LIN {X 0,Y 573.249,Z 308.076,A -85,B 0,C 180,E1 -2303.077,E2 -2303.077} C_VEL
LIN {X 0,Y 573.266,Z 308.08,A -85,B 0,C 180,E1 -2305.671,E2 -2305.671} C_VEL
LIN {X 0,Y 573.24,Z 308.077,A -85,B 0,C 180,E1 -2308.184,E2 -2308.184} C_VEL
LIN {X 0,Y 573.229,Z 308.083,A -85,B 0,C 180,E1 -2310.632,E2 -2310.632} C_VEL
LIN {X 0,Y 573.245,Z 308.077,A -85,B 0,C 180,E1 -2313.809,E2 -2313.809} C_VEL
LIN {X 0,Y 573.224,Z 308.085,A -85,B 0,C 180,E1 -2316.134,E2 -2316.134} C_VEL
LIN {X 0,Y 573.253,Z 308.079,A -85,B 0,C 180,E1 -2319.174,E2 -2319.174} C_VEL
LIN {X 0,Y 573.227,Z 308.083,A -85,B 0,C 180,E1 -2321.411,E2 -2321.411} C_VEL
LIN {X 0,Y 573.228,Z 308.079,A -85,B 0,C 180,E1 -2323.621,E2 -2323.621} C_VEL
LIN {X 0,Y 573.243,Z 308.078,A -85,B 0,C 180,E1 -2325.806,E2 -2325.806} C_VEL
LIN {X 0,Y 573.251,Z 308.075,A -85,B 0,C 180,E1 -2328.745,E2 -2328.745} C_VEL
LIN {X 0,Y 573.299,Z 308.076,A -85,B 0,C 180,E1 -2331.541,E2 -2331.541} C_VEL
LIN {X 0,Y 573.299,Z 308.071,A -85,B 0,C 180,E1 -2334.372,E2 -2334.372} C_VEL
LIN {X 0,Y 573.306,Z 308.071,A -85,B 0,C 180,E1 -2337.892,E2 -2337.892} C_VEL
LIN {X 0,Y 573.301,Z 308.069,A -85,B 0,C 180,E1 -2340.702,E2 -2340.702} C_VEL
LIN {X 0,Y 573.286,Z 308.071,A -85,B 0,C 180,E1 -2342.811,E2 -2342.811} C_VEL
LIN {X 0,Y 573.299,Z 308.071,A -85,B 0,C 180,E1 -2345.628,E2 -2345.628} C_VEL
LIN {X 0,Y 573.299,Z 308.076,A -85,B 0,C 180,E1 -2348.459,E2 -2348.459} C_VEL
LIN {X 0,Y 573.26,Z 308.075,A -85,B 0,C 180,E1 -2351.312,E2 -2351.312} C_VEL
LIN {X 0,Y 573.254,Z 308.075,A -85,B 0,C 180,E1 -2354.419,E2 -2354.419} C_VEL
LIN {X 0,Y 573.248,Z 308.083,A -85,B 0,C 180,E1 -2357.112,E2 -2357.112} C_VEL
LIN {X 0,Y 573.249,Z 308.077,A -85,B 0,C 180,E1 -2360.077,E2 -2360.077} C_VEL
LIN {X 0,Y 573.23,Z 308.085,A -85,B 0,C 180,E1 -2362.338,E2 -2362.338} C_VEL
LIN {X 0,Y 573.242,Z 308.078,A -85,B 0,C 180,E1 -2364.396,E2 -2364.396} C_VEL
LIN {X 0,Y 572.612,Z 308.156,A -85,B 0,C 180,E1 -2364.982,E2 -2364.982} C_VEL
LIN {X 0,Y 569.758,Z 308.518,A -85,B 0,C 180,E1 -2365.933,E2 -2365.933} C_VEL
LIN {X 0,Y 567.31,Z 308.826,A -85,B 0,C 180,E1 -2366.699,E2 -2366.699} C_VEL
LIN {X 0,Y 566.241,Z 308.956,A -85,B 0,C 180,E1 -2367.29,E2 -2367.29} C_VEL
LIN {X 0,Y 566.146,Z 308.965,A -85,B 0,C 180,E1 -2367.49,E2 -2367.49} C_VEL
LIN {X 0,Y 566.162,Z 308.959,A -85,B 0,C 180,E1 -2369.771,E2 -2369.771} C_VEL
LIN {X 0,Y 566.2,Z 308.959,A -85,B 0,C 180,E1 -2372.432,E2 -2372.432} C_VEL
LIN {X 0,Y 566.205,Z 308.954,A -85,B 0,C 180,E1 -2374.995,E2 -2374.995} C_VEL
LIN {X 0,Y 566.189,Z 308.96,A -85,B 0,C 180,E1 -2377.462,E2 -2377.462} C_VEL
LIN {X 0,Y 566.2,Z 308.954,A -85,B 0,C 180,E1 -2380.2,E2 -2380.2} C_VEL
LIN {X 0,Y 566.175,Z 308.961,A -85,B 0,C 180,E1 -2383.057,E2 -2383.057} C_VEL
LIN {X 0,Y 566.194,Z 308.958,A -85,B 0,C 180,E1 -2386.05,E2 -2386.05} C_VEL
LIN {X 0,Y 566.208,Z 308.953,A -85,B 0,C 180,E1 -2388.865,E2 -2388.865} C_VEL
LIN {X 0,Y 566.184,Z 308.961,A -85,B 0,C 180,E1 -2391.638,E2 -2391.638} C_VEL
LIN {X 0,Y 566.132,Z 308.964,A -85,B 0,C 180,E1 -2394.307,E2 -2394.307} C_VEL
LIN {X 0,Y 566.172,Z 309.762,A -85,B 0,C 180,E1 -2395.181,E2 -2395.181} C_VEL
LIN {X 0,Y 566.158,Z 313.905,A -85,B 0,C 180,E1 -2397.74,E2 -2397.74} C_VEL
LIN {X 0,Y 566.063,Z 318.167,A -85,B 0,C 180,E1 -2400.354,E2 -2400.354} C_VEL
LIN {X 0,Y 566.044,Z 322,A -85,B 0,C 180,E1 -2402.653,E2 -2402.653} C_VEL
LIN {X 0,Y 566.04,Z 326.033,A -85,B 0,C 180,E1 -2405.031,E2 -2405.031} C_VEL
LIN {X 0,Y 565.976,Z 330.049,A -85,B 0,C 180,E1 -2407.361,E2 -2407.361} C_VEL
LIN {X 0,Y 565.93,Z 334.103,A -85,B 0,C 180,E1 -2409.653,E2 -2409.653} C_VEL
LIN {X 0,Y 565.903,Z 338.25,A -85,B 0,C 180,E1 -2411.913,E2 -2411.913} C_VEL
LIN {X 0,Y 565.913,Z 343.78,A -85,B 0,C 180,E1 -2414.883,E2 -2414.883} C_VEL
LIN {X 0,Y 565.889,Z 348.532,A -85,B 0,C 180,E1 -2417.402,E2 -2417.402} C_VEL
LIN {X 0,Y 566.917,Z 355.474,A -85,B 0,C 180,E1 -2417.585,E2 -2417.585} C_VEL
LIN {X 0,Y 566.768,Z 368.5,A -85,B 0,C 180,E1 -2417.968,E2 -2417.968} C_VEL
LIN {X 0,Y 566.608,Z 381.072,A -85,B 0,C 180,E1 -2418.491,E2 -2418.491} C_VEL
LIN {X 0,Y 566.531,Z 392.345,A -85,B 0,C 180,E1 -2419.114,E2 -2419.114} C_VEL
LIN {X 0,Y 566.404,Z 403.688,A -85,B 0,C 180,E1 -2419.906,E2 -2419.906} C_VEL
LIN {X 0,Y 566.255,Z 413.063,A -85,B 0,C 180,E1 -2420.715,E2 -2420.715} C_VEL
LIN {X 0,Y 566.158,Z 421.62,A -85,B 0,C 180,E1 -2421.613,E2 -2421.613} C_VEL
LIN {X 0,Y 566.063,Z 429.931,A -85,B 0,C 180,E1 -2422.689,E2 -2422.689} C_VEL
LIN {X 0,Y 565.988,Z 436.626,A -85,B 0,C 180,E1 -2423.763,E2 -2423.763} C_VEL
LIN {X 0,Y 565.877,Z 442.766,A -85,B 0,C 180,E1 -2425.013,E2 -2425.013} C_VEL
LIN {X 0,Y 565.926,Z 446.755,A -85,B 0,C 180,E1 -2426.084,E2 -2426.084} C_VEL
LIN {X 0,Y 565.877,Z 449.703,A -85,B 0,C 180,E1 -2427.153,E2 -2427.153} C_VEL
LIN {X 0,Y 565.841,Z 451.128,A -85,B 0,C 180,E1 -2427.865,E2 -2427.865} C_VEL
LIN {X 0,Y 565.841,Z 452.756,A -85,B 0,C 180,E1 -2429.289,E2 -2429.289} C_VEL
LIN {X 0,Y 565.839,Z 452.996,A -85,B 0,C 180,E1 -2430,E2 -2430} C_VEL
LIN {X 0,Y 565.841,Z 452.814,A -85,B 0,C 180,E1 -2430.712,E2 -2430.712} C_VEL
LIN {X 0,Y 565.841,Z 451.268,A -85,B 0,C 180,E1 -2432.136,E2 -2432.136} C_VEL
LIN {X 0,Y 565.878,Z 449.907,A -85,B 0,C 180,E1 -2432.848,E2 -2432.848} C_VEL
LIN {X 0,Y 565.926,Z 447.029,A -85,B 0,C 180,E1 -2433.917,E2 -2433.917} C_VEL
LIN {X 0,Y 565.878,Z 443.128,A -85,B 0,C 180,E1 -2434.988,E2 -2434.988} C_VEL
LIN {X 0,Y 565.991,Z 438.096,A -85,B 0,C 180,E1 -2436.059,E2 -2436.059} C_VEL
LIN {X 0,Y 566.031,Z 431.771,A -85,B 0,C 180,E1 -2437.133,E2 -2437.133} C_VEL
LIN {X 0,Y 566.128,Z 423.849,A -85,B 0,C 180,E1 -2438.208,E2 -2438.208} C_VEL
LIN {X 0,Y 566.249,Z 413.997,A -85,B 0,C 180,E1 -2439.285,E2 -2439.285} C_VEL
LIN {X 0,Y 566.418,Z 403.677,A -85,B 0,C 180,E1 -2440.184,E2 -2440.184} C_VEL
LIN {X 0,Y 566.512,Z 392.541,A -85,B 0,C 180,E1 -2440.964,E2 -2440.964} C_VEL
LIN {X 0,Y 566.624,Z 381.186,A -85,B 0,C 180,E1 -2441.593,E2 -2441.593} C_VEL
LIN {X 0,Y 566.785,Z 368.591,A -85,B 0,C 180,E1 -2442.119,E2 -2442.119} C_VEL
LIN {X 0,Y 566.926,Z 355.415,A -85,B 0,C 180,E1 -2442.507,E2 -2442.507} C_VEL
LIN {X 0,Y 565.892,Z 348.529,A -85,B 0,C 180,E1 -2442.69,E2 -2442.69} C_VEL
LIN {X 0,Y 565.912,Z 343.948,A -85,B 0,C 180,E1 -2445.117,E2 -2445.117} C_VEL
LIN {X 0,Y 565.895,Z 338.415,A -85,B 0,C 180,E1 -2448.088,E2 -2448.088} C_VEL
LIN {X 0,Y 565.93,Z 334.266,A -85,B 0,C 180,E1 -2450.348,E2 -2450.348} C_VEL
LIN {X 0,Y 566,Z 328.864,A -85,B 0,C 180,E1 -2453.412,E2 -2453.412} C_VEL
LIN {X 0,Y 566.016,Z 324.851,A -85,B 0,C 180,E1 -2455.758,E2 -2455.758} C_VEL
LIN {X 0,Y 566.084,Z 320.751,A -85,B 0,C 180,E1 -2458.179,E2 -2458.179} C_VEL
LIN {X 0,Y 566.113,Z 315.404,A -85,B 0,C 180,E1 -2461.426,E2 -2461.426} C_VEL
LIN {X 0,Y 566.183,Z 311.295,A -85,B 0,C 180,E1 -2463.957,E2 -2463.957} C_VEL
LIN {X 0,Y 566.156,Z 309.642,A -85,B 0,C 180,E1 -2464.985,E2 -2464.985} C_VEL
LIN {X 0,Y 566.133,Z 308.964,A -85,B 0,C 180,E1 -2465.694,E2 -2465.694} C_VEL
LIN {X 0,Y 566.206,Z 308.96,A -85,B 0,C 180,E1 -2468.557,E2 -2468.557} C_VEL
LIN {X 0,Y 566.182,Z 308.956,A -85,B 0,C 180,E1 -2471.138,E2 -2471.138} C_VEL
LIN {X 0,Y 566.197,Z 308.958,A -85,B 0,C 180,E1 -2474.035,E2 -2474.035} C_VEL
LIN {X 0,Y 566.182,Z 308.961,A -85,B 0,C 180,E1 -2477.084,E2 -2477.084} C_VEL
LIN {X 0,Y 566.202,Z 308.954,A -85,B 0,C 180,E1 -2479.8,E2 -2479.8} C_VEL
LIN {X 0,Y 566.195,Z 308.959,A -85,B 0,C 180,E1 -2482.599,E2 -2482.599} C_VEL
LIN {X 0,Y 566.207,Z 308.954,A -85,B 0,C 180,E1 -2485.182,E2 -2485.182} C_VEL
LIN {X 0,Y 566.232,Z 308.954,A -85,B 0,C 180,E1 -2487.743,E2 -2487.743} C_VEL
LIN {X 0,Y 566.167,Z 308.958,A -85,B 0,C 180,E1 -2490.333,E2 -2490.333} C_VEL
LIN {X 0,Y 566.181,Z 308.957,A -85,B 0,C 180,E1 -2493.457,E2 -2493.457} C_VEL
LIN {X 0,Y 566.174,Z 308.961,A -85,B 0,C 180,E1 -2495.818,E2 -2495.818} C_VEL
LIN {X 0,Y 566.213,Z 308.953,A -85,B 0,C 180,E1 -2498.902,E2 -2498.902} C_VEL
LIN {X 0,Y 566.2,Z 308.961,A -85,B 0,C 180,E1 -2501.172,E2 -2501.172} C_VEL
LIN {X 0,Y 566.202,Z 308.954,A -85,B 0,C 180,E1 -2503.412,E2 -2503.412} C_VEL
LIN {X 0,Y 566.163,Z 308.965,A -85,B 0,C 180,E1 -2506.358,E2 -2506.358} C_VEL
LIN {X 0,Y 566.231,Z 308.952,A -85,B 0,C 180,E1 -2509.27,E2 -2509.27} C_VEL
LIN {X 0,Y 566.232,Z 308.951,A -85,B 0,C 180,E1 -2512.153,E2 -2512.153} C_VEL
LIN {X 0,Y 566.275,Z 308.95,A -85,B 0,C 180,E1 -2515.016,E2 -2515.016} C_VEL
LIN {X 0,Y 566.279,Z 308.945,A -85,B 0,C 180,E1 -2517.866,E2 -2517.866} C_VEL
LIN {X 0,Y 566.277,Z 308.945,A -85,B 0,C 180,E1 -2520.711,E2 -2520.711} C_VEL
LIN {X 0,Y 566.255,Z 308.948,A -85,B 0,C 180,E1 -2522.846,E2 -2522.846} C_VEL
LIN {X 0,Y 566.269,Z 308.947,A -85,B 0,C 180,E1 -2525.698,E2 -2525.698} C_VEL
LIN {X 0,Y 566.243,Z 308.955,A -85,B 0,C 180,E1 -2528.565,E2 -2528.565} C_VEL
LIN {X 0,Y 566.235,Z 308.95,A -85,B 0,C 180,E1 -2531.454,E2 -2531.454} C_VEL
LIN {X 0,Y 566.204,Z 308.954,A -85,B 0,C 180,E1 -2534.497,E2 -2534.497} C_VEL
LIN {X 0,Y 566.193,Z 308.96,A -85,B 0,C 180,E1 -2537.332,E2 -2537.332} C_VEL
LIN {X 0,Y 566.215,Z 308.956,A -85,B 0,C 180,E1 -2540.337,E2 -2540.337} C_VEL
LIN {X 0,Y 566.185,Z 308.956,A -85,B 0,C 180,E1 -2543.404,E2 -2543.404} C_VEL
LIN {X 0,Y 566.195,Z 308.961,A -85,B 0,C 180,E1 -2545.75,E2 -2545.75} C_VEL
LIN {X 0,Y 566.142,Z 308.961,A -85,B 0,C 180,E1 -2548.192,E2 -2548.192} C_VEL
LIN {X 0,Y 566.188,Z 308.96,A -85,B 0,C 180,E1 -2551.077,E2 -2551.077} C_VEL
LIN {X 0,Y 566.208,Z 308.954,A -85,B 0,C 180,E1 -2553.735,E2 -2553.735} C_VEL
LIN {X 0,Y 566.212,Z 308.953,A -85,B 0,C 180,E1 -2556.569,E2 -2556.569} C_VEL
LIN {X 0,Y 566.207,Z 308.956,A -85,B 0,C 180,E1 -2559.686,E2 -2559.686} C_VEL
LIN {X 0,Y 566.166,Z 308.958,A -85,B 0,C 180,E1 -2562.092,E2 -2562.092} C_VEL
LIN {X 0,Y 566.165,Z 308.96,A -85,B 0,C 180,E1 -2565.037,E2 -2565.037} C_VEL
LIN {X 0,Y 566.217,Z 308.958,A -85,B 0,C 180,E1 -2568.136,E2 -2568.136} C_VEL
LIN {X 0,Y 566.212,Z 308.954,A -85,B 0,C 180,E1 -2570.727,E2 -2570.727} C_VEL
LIN {X 0,Y 566.204,Z 309.051,A -85,B 0,C 180,E1 -2573.482,E2 -2573.482} C_VEL
LIN {X 0,Y 566.571,Z 312.745,A -85,B 0,C 180,E1 -2574.954,E2 -2574.954} C_VEL
LIN {X 0,Y 566.458,Z 320.074,A -85,B 0,C 180,E1 -2577.758,E2 -2577.758} C_VEL
LIN {X 0,Y 566.418,Z 327.929,A -85,B 0,C 180,E1 -2580.676,E2 -2580.676} C_VEL
LIN {X 0,Y 566.293,Z 336.77,A -85,B 0,C 180,E1 -2583.86,E2 -2583.86} C_VEL
LIN {X 0,Y 566.196,Z 344.898,A -85,B 0,C 180,E1 -2586.714,E2 -2586.714} C_VEL
LIN {X 0,Y 566.146,Z 352.352,A -85,B 0,C 180,E1 -2589.281,E2 -2589.281} C_VEL
LIN {X 0,Y 566.071,Z 360.144,A -85,B 0,C 180,E1 -2591.918,E2 -2591.918} C_VEL
LIN {X 0,Y 566.028,Z 367.935,A -85,B 0,C 180,E1 -2594.517,E2 -2594.517} C_VEL
LIN {X 0,Y 565.978,Z 376.491,A -85,B 0,C 180,E1 -2597.335,E2 -2597.335} C_VEL
LIN {X 0,Y 566.951,Z 383.507,A -85,B 0,C 180,E1 -2597.494,E2 -2597.494} C_VEL
LIN {X 0,Y 566.826,Z 395.875,A -85,B 0,C 180,E1 -2597.832,E2 -2597.832} C_VEL
LIN {X 0,Y 566.645,Z 408.898,A -85,B 0,C 180,E1 -2598.346,E2 -2598.346} C_VEL
LIN {X 0,Y 566.54,Z 420.385,A -85,B 0,C 180,E1 -2598.949,E2 -2598.949} C_VEL
LIN {X 0,Y 566.442,Z 431.928,A -85,B 0,C 180,E1 -2599.726,E2 -2599.726} C_VEL
LIN {X 0,Y 566.282,Z 441.599,A -85,B 0,C 180,E1 -2600.535,E2 -2600.535} C_VEL
LIN {X 0,Y 566.181,Z 450.412,A -85,B 0,C 180,E1 -2601.433,E2 -2601.433} C_VEL
LIN {X 0,Y 566.056,Z 458.999,A -85,B 0,C 180,E1 -2602.509,E2 -2602.509} C_VEL
LIN {X 0,Y 565.965,Z 465.866,A -85,B 0,C 180,E1 -2603.583,E2 -2603.583} C_VEL
LIN {X 0,Y 565.937,Z 471.364,A -85,B 0,C 180,E1 -2604.656,E2 -2604.656} C_VEL
LIN {X 0,Y 565.959,Z 475.676,A -85,B 0,C 180,E1 -2605.727,E2 -2605.727} C_VEL
LIN {X 0,Y 565.927,Z 477.956,A -85,B 0,C 180,E1 -2606.44,E2 -2606.44} C_VEL
LIN {X 0,Y 565.878,Z 479.808,A -85,B 0,C 180,E1 -2607.152,E2 -2607.152} C_VEL
LIN {X 0,Y 565.841,Z 481.2,A -85,B 0,C 180,E1 -2607.864,E2 -2607.864} C_VEL
LIN {X 0,Y 565.841,Z 482.784,A -85,B 0,C 180,E1 -2609.288,E2 -2609.288} C_VEL
LIN {X 0,Y 565.839,Z 483,A -85,B 0,C 180,E1 -2610,E2 -2610} C_VEL
LIN {X 0,Y 565.846,Z 482.186,A -85,B 0,C 180,E1 -2611.423,E2 -2611.423} C_VEL
LIN {X 0,Y 565.841,Z 481.201,A -85,B 0,C 180,E1 -2612.135,E2 -2612.135} C_VEL
LIN {X 0,Y 565.878,Z 479.811,A -85,B 0,C 180,E1 -2612.847,E2 -2612.847} C_VEL
LIN {X 0,Y 565.926,Z 476.897,A -85,B 0,C 180,E1 -2613.916,E2 -2613.916} C_VEL
LIN {X 0,Y 565.878,Z 472.951,A -85,B 0,C 180,E1 -2614.987,E2 -2614.987} C_VEL
LIN {X 0,Y 566.002,Z 467.869,A -85,B 0,C 180,E1 -2616.058,E2 -2616.058} C_VEL
LIN {X 0,Y 566.04,Z 461.473,A -85,B 0,C 180,E1 -2617.132,E2 -2617.132} C_VEL
LIN {X 0,Y 566.133,Z 453.482,A -85,B 0,C 180,E1 -2618.207,E2 -2618.207} C_VEL
LIN {X 0,Y 566.228,Z 445.342,A -85,B 0,C 180,E1 -2619.105,E2 -2619.105} C_VEL
LIN {X 0,Y 566.344,Z 435.408,A -85,B 0,C 180,E1 -2620.004,E2 -2620.004} C_VEL
LIN {X 0,Y 566.5,Z 424.336,A -85,B 0,C 180,E1 -2620.805,E2 -2620.805} C_VEL
LIN {X 0,Y 566.607,Z 411.962,A -85,B 0,C 180,E1 -2621.509,E2 -2621.509} C_VEL
LIN {X 0,Y 566.748,Z 399.783,A -85,B 0,C 180,E1 -2622.033,E2 -2622.033} C_VEL
LIN {X 0,Y 566.912,Z 386.373,A -85,B 0,C 180,E1 -2622.438,E2 -2622.438} C_VEL
LIN {X 0,Y 566.642,Z 380.688,A -85,B 0,C 180,E1 -2622.569,E2 -2622.569} C_VEL
LIN {X 0,Y 565.978,Z 376.493,A -85,B 0,C 180,E1 -2622.664,E2 -2622.664} C_VEL
LIN {X 0,Y 566.027,Z 367.937,A -85,B 0,C 180,E1 -2625.482,E2 -2625.482} C_VEL
LIN {X 0,Y 566.086,Z 359.033,A -85,B 0,C 180,E1 -2628.456,E2 -2628.456} C_VEL
LIN {X 0,Y 566.199,Z 350.309,A -85,B 0,C 180,E1 -2631.417,E2 -2631.417} C_VEL
LIN {X 0,Y 566.258,Z 341.224,A -85,B 0,C 180,E1 -2634.567,E2 -2634.567} C_VEL
LIN {X 0,Y 566.327,Z 333.433,A -85,B 0,C 180,E1 -2637.332,E2 -2637.332} C_VEL
LIN {X 0,Y 566.408,Z 325.642,A -85,B 0,C 180,E1 -2640.166,E2 -2640.166} C_VEL
LIN {X 0,Y 566.48,Z 319.458,A -85,B 0,C 180,E1 -2642.473,E2 -2642.473} C_VEL
LIN {X 0,Y 566.581,Z 312.739,A -85,B 0,C 180,E1 -2645.047,E2 -2645.047} C_VEL
LIN {X 0,Y 566.211,Z 308.96,A -85,B 0,C 180,E1 -2646.568,E2 -2646.568} C_VEL
LIN {X 0,Y 566.208,Z 308.955,A -85,B 0,C 180,E1 -2649.685,E2 -2649.685} C_VEL
LIN {X 0,Y 566.21,Z 308.96,A -85,B 0,C 180,E1 -2652.086,E2 -2652.086} C_VEL
LIN {X 0,Y 566.168,Z 308.96,A -85,B 0,C 180,E1 -2655.035,E2 -2655.035} C_VEL
LIN {X 0,Y 566.164,Z 308.958,A -85,B 0,C 180,E1 -2657.908,E2 -2657.908} C_VEL
LIN {X 0,Y 566.208,Z 308.958,A -85,B 0,C 180,E1 -2660.726,E2 -2660.726} C_VEL
LIN {X 0,Y 566.211,Z 308.957,A -85,B 0,C 180,E1 -2663.783,E2 -2663.783} C_VEL
LIN {X 0,Y 566.204,Z 308.955,A -85,B 0,C 180,E1 -2666.265,E2 -2666.265} C_VEL
LIN {X 0,Y 566.185,Z 308.96,A -85,B 0,C 180,E1 -2668.922,E2 -2668.922} C_VEL
LIN {X 0,Y 566.14,Z 308.961,A -85,B 0,C 180,E1 -2671.853,E2 -2671.853} C_VEL
LIN {X 0,Y 566.198,Z 308.961,A -85,B 0,C 180,E1 -2674.25,E2 -2674.25} C_VEL
LIN {X 0,Y 566.182,Z 308.956,A -85,B 0,C 180,E1 -2676.713,E2 -2676.713} C_VEL
LIN {X 0,Y 566.211,Z 308.957,A -85,B 0,C 180,E1 -2679.663,E2 -2679.663} C_VEL
LIN {X 0,Y 566.192,Z 308.96,A -85,B 0,C 180,E1 -2682.668,E2 -2682.668} C_VEL
LIN {X 0,Y 566.206,Z 308.953,A -85,B 0,C 180,E1 -2685.626,E2 -2685.626} C_VEL
LIN {X 0,Y 566.223,Z 308.951,A -85,B 0,C 180,E1 -2688.675,E2 -2688.675} C_VEL
LIN {X 0,Y 566.239,Z 308.956,A -85,B 0,C 180,E1 -2691.434,E2 -2691.434} C_VEL
LIN {X 0,Y 566.266,Z 308.947,A -85,B 0,C 180,E1 -2694.302,E2 -2694.302} C_VEL
LIN {X 0,Y 566.276,Z 308.947,A -85,B 0,C 180,E1 -2697.866,E2 -2697.866} C_VEL
LIN {X 0,Y 566.274,Z 308.945,A -85,B 0,C 180,E1 -2700.711,E2 -2700.711} C_VEL
LIN {X 0,Y 566.254,Z 308.947,A -85,B 0,C 180,E1 -2702.846,E2 -2702.846} C_VEL
LIN {X 0,Y 566.266,Z 308.947,A -85,B 0,C 180,E1 -2705.698,E2 -2705.698} C_VEL
LIN {X 0,Y 566.239,Z 308.955,A -85,B 0,C 180,E1 -2708.566,E2 -2708.566} C_VEL
LIN {X 0,Y 566.23,Z 308.952,A -85,B 0,C 180,E1 -2711.455,E2 -2711.455} C_VEL
LIN {X 0,Y 566.209,Z 308.953,A -85,B 0,C 180,E1 -2714.502,E2 -2714.502} C_VEL
LIN {X 0,Y 566.192,Z 308.959,A -85,B 0,C 180,E1 -2717.332,E2 -2717.332} C_VEL
LIN {X 0,Y 566.212,Z 308.957,A -85,B 0,C 180,E1 -2720.337,E2 -2720.337} C_VEL
LIN {X 0,Y 566.181,Z 308.958,A -85,B 0,C 180,E1 -2723.404,E2 -2723.404} C_VEL
LIN {X 0,Y 566.198,Z 308.96,A -85,B 0,C 180,E1 -2725.75,E2 -2725.75} C_VEL
LIN {X 0,Y 566.146,Z 308.965,A -85,B 0,C 180,E1 -2727.49,E2 -2727.49} C_VEL
LIN {X 0,Y 565.46,Z 309.048,A -85,B 0,C 180,E1 -2728.084,E2 -2728.084} C_VEL
LIN {X 0,Y 562.604,Z 309.408,A -85,B 0,C 180,E1 -2729.048,E2 -2729.048} C_VEL
LIN {X 0,Y 560.214,Z 309.702,A -85,B 0,C 180,E1 -2729.824,E2 -2729.824} C_VEL
LIN {X 0,Y 559.201,Z 309.827,A -85,B 0,C 180,E1 -2730.423,E2 -2730.423} C_VEL
LIN {X 0,Y 559.125,Z 309.836,A -85,B 0,C 180,E1 -2730.625,E2 -2730.625} C_VEL
LIN {X 0,Y 559.168,Z 309.835,A -85,B 0,C 180,E1 -2732.715,E2 -2732.715} C_VEL
LIN {X 0,Y 559.15,Z 309.833,A -85,B 0,C 180,E1 -2735.323,E2 -2735.323} C_VEL
LIN {X 0,Y 559.125,Z 309.839,A -85,B 0,C 180,E1 -2738.018,E2 -2738.018} C_VEL
LIN {X 0,Y 559.145,Z 309.836,A -85,B 0,C 180,E1 -2740.814,E2 -2740.814} C_VEL
LIN {X 0,Y 559.108,Z 309.837,A -85,B 0,C 180,E1 -2743.737,E2 -2743.737} C_VEL
LIN {X 0,Y 559.155,Z 309.838,A -85,B 0,C 180,E1 -2746.269,E2 -2746.269} C_VEL
LIN {X 0,Y 559.173,Z 309.831,A -85,B 0,C 180,E1 -2749.19,E2 -2749.19} C_VEL
LIN {X 0,Y 559.13,Z 309.836,A -85,B 0,C 180,E1 -2751.983,E2 -2751.983} C_VEL
LIN {X 0,Y 559.062,Z 309.849,A -85,B 0,C 180,E1 -2754.672,E2 -2754.672} C_VEL
LIN {X 0,Y 559.119,Z 312.614,A -85,B 0,C 180,E1 -2756.423,E2 -2756.423} C_VEL
LIN {X 0,Y 559.062,Z 316.714,A -85,B 0,C 180,E1 -2758.976,E2 -2758.976} C_VEL
LIN {X 0,Y 559.029,Z 321.058,A -85,B 0,C 180,E1 -2761.646,E2 -2761.646} C_VEL
LIN {X 0,Y 558.97,Z 326.425,A -85,B 0,C 180,E1 -2764.86,E2 -2764.86} C_VEL
LIN {X 0,Y 558.907,Z 331.524,A -85,B 0,C 180,E1 -2767.838,E2 -2767.838} C_VEL
LIN {X 0,Y 558.874,Z 336.886,A -85,B 0,C 180,E1 -2770.917,E2 -2770.917} C_VEL
LIN {X 0,Y 558.787,Z 342.399,A -85,B 0,C 180,E1 -2773.937,E2 -2773.937} C_VEL
LIN {X 0,Y 558.806,Z 346.546,A -85,B 0,C 180,E1 -2776.175,E2 -2776.175} C_VEL
LIN {X 0,Y 558.82,Z 348.533,A -85,B 0,C 180,E1 -2777.24,E2 -2777.24} C_VEL
LIN {X 0,Y 559.958,Z 356.41,A -85,B 0,C 180,E1 -2777.451,E2 -2777.451} C_VEL
LIN {X 0,Y 559.799,Z 369.812,A -85,B 0,C 180,E1 -2777.862,E2 -2777.862} C_VEL
LIN {X 0,Y 559.639,Z 382.319,A -85,B 0,C 180,E1 -2778.409,E2 -2778.409} C_VEL
LIN {X 0,Y 559.54,Z 393.735,A -85,B 0,C 180,E1 -2779.065,E2 -2779.065} C_VEL
LIN {X 0,Y 559.348,Z 404.857,A -85,B 0,C 180,E1 -2779.869,E2 -2779.869} C_VEL
LIN {X 0,Y 559.21,Z 414.9,A -85,B 0,C 180,E1 -2780.78,E2 -2780.78} C_VEL
LIN {X 0,Y 559.05,Z 424.599,A -85,B 0,C 180,E1 -2781.87,E2 -2781.87} C_VEL
LIN {X 0,Y 558.971,Z 432.459,A -85,B 0,C 180,E1 -2782.977,E2 -2782.977} C_VEL
LIN {X 0,Y 558.936,Z 439.457,A -85,B 0,C 180,E1 -2784.227,E2 -2784.227} C_VEL
LIN {X 0,Y 558.826,Z 444.197,A -85,B 0,C 180,E1 -2785.311,E2 -2785.311} C_VEL
LIN {X 0,Y 558.836,Z 447.829,A -85,B 0,C 180,E1 -2786.395,E2 -2786.395} C_VEL
LIN {X 0,Y 558.799,Z 449.705,A -85,B 0,C 180,E1 -2787.117,E2 -2787.117} C_VEL
LIN {X 0,Y 558.747,Z 451.129,A -85,B 0,C 180,E1 -2787.838,E2 -2787.838} C_VEL
LIN {X 0,Y 558.741,Z 452.757,A -85,B 0,C 180,E1 -2789.28,E2 -2789.28} C_VEL
LIN {X 0,Y 558.74,Z 452.996,A -85,B 0,C 180,E1 -2790,E2 -2790} C_VEL
LIN {X 0,Y 558.741,Z 452.814,A -85,B 0,C 180,E1 -2790.721,E2 -2790.721} C_VEL
LIN {X 0,Y 558.747,Z 451.266,A -85,B 0,C 180,E1 -2792.163,E2 -2792.163} C_VEL
LIN {X 0,Y 558.8,Z 449.905,A -85,B 0,C 180,E1 -2792.884,E2 -2792.884} C_VEL
LIN {X 0,Y 558.844,Z 447.027,A -85,B 0,C 180,E1 -2793.966,E2 -2793.966} C_VEL
LIN {X 0,Y 558.798,Z 443.126,A -85,B 0,C 180,E1 -2795.051,E2 -2795.051} C_VEL
LIN {X 0,Y 558.911,Z 438.093,A -85,B 0,C 180,E1 -2796.136,E2 -2796.136} C_VEL
LIN {X 0,Y 558.973,Z 431.767,A -85,B 0,C 180,E1 -2797.223,E2 -2797.223} C_VEL
LIN {X 0,Y 559.091,Z 423.844,A -85,B 0,C 180,E1 -2798.312,E2 -2798.312} C_VEL
LIN {X 0,Y 559.224,Z 413.991,A -85,B 0,C 180,E1 -2799.403,E2 -2799.403} C_VEL
LIN {X 0,Y 559.417,Z 403.671,A -85,B 0,C 180,E1 -2800.313,E2 -2800.313} C_VEL
LIN {X 0,Y 559.539,Z 392.825,A -85,B 0,C 180,E1 -2801.083,E2 -2801.083} C_VEL
LIN {X 0,Y 559.634,Z 382.272,A -85,B 0,C 180,E1 -2801.683,E2 -2801.683} C_VEL
LIN {X 0,Y 559.838,Z 369.741,A -85,B 0,C 180,E1 -2802.23,E2 -2802.23} C_VEL
LIN {X 0,Y 559.989,Z 356.307,A -85,B 0,C 180,E1 -2802.641,E2 -2802.641} C_VEL
LIN {X 0,Y 558.79,Z 348.528,A -85,B 0,C 180,E1 -2802.854,E2 -2802.854} C_VEL
LIN {X 0,Y 558.825,Z 343.946,A -85,B 0,C 180,E1 -2805.314,E2 -2805.314} C_VEL
LIN {X 0,Y 558.811,Z 338.414,A -85,B 0,C 180,E1 -2808.326,E2 -2808.326} C_VEL
LIN {X 0,Y 558.856,Z 334.399,A -85,B 0,C 180,E1 -2810.617,E2 -2810.617} C_VEL
LIN {X 0,Y 558.931,Z 329.574,A -85,B 0,C 180,E1 -2813.378,E2 -2813.378} C_VEL
LIN {X 0,Y 558.942,Z 324.962,A -85,B 0,C 180,E1 -2816.109,E2 -2816.109} C_VEL
LIN {X 0,Y 559.027,Z 320.906,A -85,B 0,C 180,E1 -2818.537,E2 -2818.537} C_VEL
LIN {X 0,Y 559.071,Z 316.48,A -85,B 0,C 180,E1 -2821.26,E2 -2821.26} C_VEL
LIN {X 0,Y 559.144,Z 312.165,A -85,B 0,C 180,E1 -2823.945,E2 -2823.945} C_VEL
LIN {X 0,Y 559.085,Z 309.973,A -85,B 0,C 180,E1 -2825.327,E2 -2825.327} C_VEL
LIN {X 0,Y 559.128,Z 309.836,A -85,B 0,C 180,E1 -2828.018,E2 -2828.018} C_VEL
LIN {X 0,Y 559.159,Z 309.833,A -85,B 0,C 180,E1 -2830.812,E2 -2830.812} C_VEL
LIN {X 0,Y 559.159,Z 309.837,A -85,B 0,C 180,E1 -2833.732,E2 -2833.732} C_VEL
LIN {X 0,Y 559.125,Z 309.837,A -85,B 0,C 180,E1 -2836.805,E2 -2836.805} C_VEL
LIN {X 0,Y 559.149,Z 309.837,A -85,B 0,C 180,E1 -2839.187,E2 -2839.187} C_VEL
LIN {X 0,Y 559.126,Z 309.838,A -85,B 0,C 180,E1 -2841.982,E2 -2841.982} C_VEL
LIN {X 0,Y 559.146,Z 309.833,A -85,B 0,C 180,E1 -2844.784,E2 -2844.784} C_VEL
LIN {X 0,Y 559.172,Z 309.835,A -85,B 0,C 180,E1 -2847.361,E2 -2847.361} C_VEL
LIN {X 0,Y 559.117,Z 309.836,A -85,B 0,C 180,E1 -2850.147,E2 -2850.147} C_VEL
LIN {X 0,Y 559.117,Z 309.838,A -85,B 0,C 180,E1 -2853.182,E2 -2853.182} C_VEL
LIN {X 0,Y 559.122,Z 309.837,A -85,B 0,C 180,E1 -2855.493,E2 -2855.493} C_VEL
LIN {X 0,Y 559.174,Z 309.83,A -85,B 0,C 180,E1 -2858.624,E2 -2858.624} C_VEL
LIN {X 0,Y 559.161,Z 309.834,A -85,B 0,C 180,E1 -2860.926,E2 -2860.926} C_VEL
LIN {X 0,Y 559.15,Z 309.832,A -85,B 0,C 180,E1 -2863.947,E2 -2863.947} C_VEL
LIN {X 0,Y 559.141,Z 309.838,A -85,B 0,C 180,E1 -2866.183,E2 -2866.183} C_VEL
LIN {X 0,Y 559.188,Z 309.828,A -85,B 0,C 180,E1 -2869.133,E2 -2869.133} C_VEL
LIN {X 0,Y 559.201,Z 309.827,A -85,B 0,C 180,E1 -2872.053,E2 -2872.053} C_VEL
LIN {X 0,Y 559.25,Z 309.826,A -85,B 0,C 180,E1 -2874.953,E2 -2874.953} C_VEL
LIN {X 0,Y 559.249,Z 309.82,A -85,B 0,C 180,E1 -2877.839,E2 -2877.839} C_VEL
LIN {X 0,Y 559.249,Z 309.82,A -85,B 0,C 180,E1 -2880.72,E2 -2880.72} C_VEL
LIN {X 0,Y 559.223,Z 309.824,A -85,B 0,C 180,E1 -2882.881,E2 -2882.881} C_VEL
LIN {X 0,Y 559.238,Z 309.823,A -85,B 0,C 180,E1 -2885.77,E2 -2885.77} C_VEL
LIN {X 0,Y 559.198,Z 309.832,A -85,B 0,C 180,E1 -2888.674,E2 -2888.674} C_VEL
LIN {X 0,Y 559.197,Z 309.828,A -85,B 0,C 180,E1 -2891.601,E2 -2891.601} C_VEL
LIN {X 0,Y 559.152,Z 309.832,A -85,B 0,C 180,E1 -2894.579,E2 -2894.579} C_VEL
LIN {X 0,Y 559.153,Z 309.835,A -85,B 0,C 180,E1 -2897.557,E2 -2897.557} C_VEL
LIN {X 0,Y 559.168,Z 309.831,A -85,B 0,C 180,E1 -2899.838,E2 -2899.838} C_VEL
LIN {X 0,Y 559.139,Z 309.839,A -85,B 0,C 180,E1 -2902.153,E2 -2902.153} C_VEL
LIN {X 0,Y 559.174,Z 309.83,A -85,B 0,C 180,E1 -2905.187,E2 -2905.187} C_VEL
LIN {X 0,Y 559.101,Z 309.842,A -85,B 0,C 180,E1 -2907.717,E2 -2907.717} C_VEL
LIN {X 0,Y 559.134,Z 309.835,A -85,B 0,C 180,E1 -2910.184,E2 -2910.184} C_VEL
LIN {X 0,Y 559.17,Z 309.836,A -85,B 0,C 180,E1 -2912.714,E2 -2912.714} C_VEL
LIN {X 0,Y 559.145,Z 309.834,A -85,B 0,C 180,E1 -2915.323,E2 -2915.323} C_VEL
LIN {X 0,Y 559.127,Z 309.838,A -85,B 0,C 180,E1 -2918.018,E2 -2918.018} C_VEL
LIN {X 0,Y 559.149,Z 309.835,A -85,B 0,C 180,E1 -2920.813,E2 -2920.813} C_VEL
LIN {X 0,Y 559.105,Z 309.838,A -85,B 0,C 180,E1 -2923.738,E2 -2923.738} C_VEL
LIN {X 0,Y 559.137,Z 309.841,A -85,B 0,C 180,E1 -2926.266,E2 -2926.266} C_VEL
LIN {X 0,Y 559.167,Z 309.831,A -85,B 0,C 180,E1 -2928.949,E2 -2928.949} C_VEL
LIN {X 0,Y 559.172,Z 309.835,A -85,B 0,C 180,E1 -2931.192,E2 -2931.192} C_VEL
LIN {X 0,Y 559.192,Z 309.998,A -85,B 0,C 180,E1 -2933.342,E2 -2933.342} C_VEL
LIN {X 0,Y 559.561,Z 313.427,A -85,B 0,C 180,E1 -2934.725,E2 -2934.725} C_VEL
LIN {X 0,Y 559.49,Z 320.086,A -85,B 0,C 180,E1 -2937.312,E2 -2937.312} C_VEL
LIN {X 0,Y 559.399,Z 327.465,A -85,B 0,C 180,E1 -2940.098,E2 -2940.098} C_VEL
LIN {X 0,Y 559.275,Z 335.791,A -85,B 0,C 180,E1 -2943.152,E2 -2943.152} C_VEL
LIN {X 0,Y 559.205,Z 343.448,A -85,B 0,C 180,E1 -2945.892,E2 -2945.892} C_VEL
LIN {X 0,Y 559.115,Z 352.352,A -85,B 0,C 180,E1 -2949.008,E2 -2949.008} C_VEL
LIN {X 0,Y 559.017,Z 360.144,A -85,B 0,C 180,E1 -2951.681,E2 -2951.681} C_VEL
LIN {X 0,Y 558.965,Z 367.935,A -85,B 0,C 180,E1 -2954.316,E2 -2954.316} C_VEL
LIN {X 0,Y 558.921,Z 376.491,A -85,B 0,C 180,E1 -2957.173,E2 -2957.173} C_VEL
LIN {X 0,Y 560.012,Z 384.52,A -85,B 0,C 180,E1 -2957.359,E2 -2957.359} C_VEL
LIN {X 0,Y 559.876,Z 397.305,A -85,B 0,C 180,E1 -2957.729,E2 -2957.729} C_VEL
LIN {X 0,Y 559.696,Z 408.281,A -85,B 0,C 180,E1 -2958.17,E2 -2958.17} C_VEL
LIN {X 0,Y 559.556,Z 419.761,A -85,B 0,C 180,E1 -2958.773,E2 -2958.773} C_VEL
LIN {X 0,Y 559.424,Z 430.745,A -85,B 0,C 180,E1 -2959.504,E2 -2959.504} C_VEL
LIN {X 0,Y 559.244,Z 441.599,A -85,B 0,C 180,E1 -2960.415,E2 -2960.415} C_VEL
LIN {X 0,Y 559.127,Z 450.412,A -85,B 0,C 180,E1 -2961.325,E2 -2961.325} C_VEL
LIN {X 0,Y 558.997,Z 458.999,A -85,B 0,C 180,E1 -2962.414,E2 -2962.414} C_VEL
LIN {X 0,Y 558.885,Z 466.687,A -85,B 0,C 180,E1 -2963.649,E2 -2963.649} C_VEL
LIN {X 0,Y 558.869,Z 471.365,A -85,B 0,C 180,E1 -2964.588,E2 -2964.588} C_VEL
LIN {X 0,Y 558.869,Z 475.677,A -85,B 0,C 180,E1 -2965.673,E2 -2965.673} C_VEL
LIN {X 0,Y 558.836,Z 477.956,A -85,B 0,C 180,E1 -2966.395,E2 -2966.395} C_VEL
LIN {X 0,Y 558.799,Z 479.808,A -85,B 0,C 180,E1 -2967.116,E2 -2967.116} C_VEL
LIN {X 0,Y 558.747,Z 481.199,A -85,B 0,C 180,E1 -2967.837,E2 -2967.837} C_VEL
LIN {X 0,Y 558.741,Z 482.784,A -85,B 0,C 180,E1 -2969.279,E2 -2969.279} C_VEL
LIN {X 0,Y 558.74,Z 483,A -85,B 0,C 180,E1 -2970,E2 -2970} C_VEL
LIN {X 0,Y 558.745,Z 482.186,A -85,B 0,C 180,E1 -2971.441,E2 -2971.441} C_VEL
LIN {X 0,Y 558.747,Z 481.201,A -85,B 0,C 180,E1 -2972.162,E2 -2972.162} C_VEL
LIN {X 0,Y 558.799,Z 479.811,A -85,B 0,C 180,E1 -2972.883,E2 -2972.883} C_VEL
LIN {X 0,Y 558.844,Z 476.897,A -85,B 0,C 180,E1 -2973.966,E2 -2973.966} C_VEL
LIN {X 0,Y 558.798,Z 472.951,A -85,B 0,C 180,E1 -2975.05,E2 -2975.05} C_VEL
LIN {X 0,Y 558.921,Z 467.869,A -85,B 0,C 180,E1 -2976.135,E2 -2976.135} C_VEL
LIN {X 0,Y 558.977,Z 461.472,A -85,B 0,C 180,E1 -2977.222,E2 -2977.222} C_VEL
LIN {X 0,Y 559.098,Z 453.482,A -85,B 0,C 180,E1 -2978.311,E2 -2978.311} C_VEL
LIN {X 0,Y 559.194,Z 445.342,A -85,B 0,C 180,E1 -2979.22,E2 -2979.22} C_VEL
LIN {X 0,Y 559.357,Z 435.408,A -85,B 0,C 180,E1 -2980.131,E2 -2980.131} C_VEL
LIN {X 0,Y 559.504,Z 424.446,A -85,B 0,C 180,E1 -2980.934,E2 -2980.934} C_VEL
LIN {X 0,Y 559.635,Z 412.834,A -85,B 0,C 180,E1 -2981.609,E2 -2981.609} C_VEL
LIN {X 0,Y 559.762,Z 401.002,A -85,B 0,C 180,E1 -2982.139,E2 -2982.139} C_VEL
LIN {X 0,Y 559.954,Z 388.2,A -85,B 0,C 180,E1 -2982.549,E2 -2982.549} C_VEL
LIN {X 0,Y 559.767,Z 381.83,A -85,B 0,C 180,E1 -2982.703,E2 -2982.703} C_VEL
LIN {X 0,Y 558.92,Z 376.493,A -85,B 0,C 180,E1 -2982.827,E2 -2982.827} C_VEL
LIN {X 0,Y 558.965,Z 367.937,A -85,B 0,C 180,E1 -2985.683,E2 -2985.683} C_VEL
LIN {X 0,Y 559.017,Z 360.146,A -85,B 0,C 180,E1 -2988.318,E2 -2988.318} C_VEL
LIN {X 0,Y 559.114,Z 352.354,A -85,B 0,C 180,E1 -2990.991,E2 -2990.991} C_VEL
LIN {X 0,Y 559.203,Z 343.45,A -85,B 0,C 180,E1 -2994.107,E2 -2994.107} C_VEL
LIN {X 0,Y 559.315,Z 334.546,A -85,B 0,C 180,E1 -2997.298,E2 -2997.298} C_VEL
LIN {X 0,Y 559.402,Z 326.755,A -85,B 0,C 180,E1 -3000.167,E2 -3000.167} C_VEL
LIN {X 0,Y 559.509,Z 318.963,A -85,B 0,C 180,E1 -3003.12,E2 -3003.12} C_VEL
LIN {X 0,Y 559.537,Z 312.27,A -85,B 0,C 180,E1 -3005.735,E2 -3005.735} C_VEL
LIN {X 0,Y 559.165,Z 309.837,A -85,B 0,C 180,E1 -3006.749,E2 -3006.749} C_VEL
LIN {X 0,Y 559.181,Z 309.832,A -85,B 0,C 180,E1 -3009.864,E2 -3009.864} C_VEL
LIN {X 0,Y 559.159,Z 309.833,A -85,B 0,C 180,E1 -3012.742,E2 -3012.742} C_VEL
LIN {X 0,Y 559.146,Z 309.836,A -85,B 0,C 180,E1 -3015.76,E2 -3015.76} C_VEL
LIN {X 0,Y 559.117,Z 309.836,A -85,B 0,C 180,E1 -3018.225,E2 -3018.225} C_VEL
LIN {X 0,Y 559.167,Z 309.831,A -85,B 0,C 180,E1 -3021.191,E2 -3021.191} C_VEL
LIN {X 0,Y 559.165,Z 309.835,A -85,B 0,C 180,E1 -3023.791,E2 -3023.791} C_VEL
LIN {X 0,Y 559.157,Z 309.832,A -85,B 0,C 180,E1 -3026.425,E2 -3026.425} C_VEL
LIN {X 0,Y 559.148,Z 309.838,A -85,B 0,C 180,E1 -3028.98,E2 -3028.98} C_VEL
LIN {X 0,Y 559.1,Z 309.838,A -85,B 0,C 180,E1 -3031.629,E2 -3031.629} C_VEL
LIN {X 0,Y 559.162,Z 309.832,A -85,B 0,C 180,E1 -3033.902,E2 -3033.902} C_VEL
LIN {X 0,Y 559.147,Z 309.834,A -85,B 0,C 180,E1 -3036.567,E2 -3036.567} C_VEL
LIN {X 0,Y 559.177,Z 309.834,A -85,B 0,C 180,E1 -3039.395,E2 -3039.395} C_VEL
LIN {X 0,Y 559.143,Z 309.835,A -85,B 0,C 180,E1 -3041.686,E2 -3041.686} C_VEL
LIN {X 0,Y 559.145,Z 309.834,A -85,B 0,C 180,E1 -3043.947,E2 -3043.947} C_VEL
LIN {X 0,Y 559.145,Z 309.839,A -85,B 0,C 180,E1 -3046.183,E2 -3046.183} C_VEL
LIN {X 0,Y 559.184,Z 309.828,A -85,B 0,C 180,E1 -3049.133,E2 -3049.133} C_VEL
LIN {X 0,Y 559.201,Z 309.827,A -85,B 0,C 180,E1 -3052.054,E2 -3052.054} C_VEL
LIN {X 0,Y 559.247,Z 309.826,A -85,B 0,C 180,E1 -3054.953,E2 -3054.953} C_VEL
LIN {X 0,Y 559.246,Z 309.822,A -85,B 0,C 180,E1 -3057.839,E2 -3057.839} C_VEL
LIN {X 0,Y 559.246,Z 309.82,A -85,B 0,C 180,E1 -3060.72,E2 -3060.72} C_VEL
LIN {X 0,Y 559.222,Z 309.824,A -85,B 0,C 180,E1 -3062.882,E2 -3062.882} C_VEL
LIN {X 0,Y 559.235,Z 309.822,A -85,B 0,C 180,E1 -3065.77,E2 -3065.77} C_VEL
LIN {X 0,Y 559.194,Z 309.833,A -85,B 0,C 180,E1 -3068.674,E2 -3068.674} C_VEL
LIN {X 0,Y 559.192,Z 309.83,A -85,B 0,C 180,E1 -3071.601,E2 -3071.601} C_VEL
LIN {X 0,Y 559.169,Z 309.83,A -85,B 0,C 180,E1 -3074.588,E2 -3074.588} C_VEL
LIN {X 0,Y 559.152,Z 309.834,A -85,B 0,C 180,E1 -3077.557,E2 -3077.557} C_VEL
LIN {X 0,Y 559.166,Z 309.831,A -85,B 0,C 180,E1 -3079.838,E2 -3079.838} C_VEL
LIN {X 0,Y 559.134,Z 309.84,A -85,B 0,C 180,E1 -3082.153,E2 -3082.153} C_VEL
LIN {X 0,Y 559.169,Z 309.832,A -85,B 0,C 180,E1 -3085.188,E2 -3085.188} C_VEL
LIN {X 0,Y 559.099,Z 309.842,A -85,B 0,C 180,E1 -3087.717,E2 -3087.717} C_VEL
LIN {X 0,Y 559.125,Z 309.836,A -85,B 0,C 180,E1 -3090.625,E2 -3090.625} C_VEL
LIN {X 0,Y 558.473,Z 309.92,A -85,B 0,C 180,E1 -3091.227,E2 -3091.227} C_VEL
LIN {X 0,Y 555.616,Z 310.275,A -85,B 0,C 180,E1 -3092.203,E2 -3092.203} C_VEL
LIN {X 0,Y 553.203,Z 310.575,A -85,B 0,C 180,E1 -3092.989,E2 -3092.989} C_VEL
LIN {X 0,Y 552.182,Z 310.701,A -85,B 0,C 180,E1 -3093.596,E2 -3093.596} C_VEL
LIN {X 0,Y 552.108,Z 310.711,A -85,B 0,C 180,E1 -3093.801,E2 -3093.801} C_VEL
LIN {X 0,Y 552.105,Z 310.711,A -85,B 0,C 180,E1 -3096.747,E2 -3096.747} C_VEL
LIN {X 0,Y 552.123,Z 310.713,A -85,B 0,C 180,E1 -3099.528,E2 -3099.528} C_VEL
LIN {X 0,Y 552.1,Z 310.713,A -85,B 0,C 180,E1 -3102.429,E2 -3102.429} C_VEL
LIN {X 0,Y 552.092,Z 310.711,A -85,B 0,C 180,E1 -3105.564,E2 -3105.564} C_VEL
LIN {X 0,Y 552.137,Z 310.707,A -85,B 0,C 180,E1 -3108.677,E2 -3108.677} C_VEL
LIN {X 0,Y 552.116,Z 310.714,A -85,B 0,C 180,E1 -3111.412,E2 -3111.412} C_VEL
LIN {X 0,Y 552.051,Z 310.718,A -85,B 0,C 180,E1 -3114.155,E2 -3114.155} C_VEL
LIN {X 0,Y 552.016,Z 310.725,A -85,B 0,C 180,E1 -3114.57,E2 -3114.57} C_VEL
LIN {X 0,Y 552.048,Z 314.08,A -85,B 0,C 180,E1 -3116.811,E2 -3116.811} C_VEL
LIN {X 0,Y 551.979,Z 318.169,A -85,B 0,C 180,E1 -3119.384,E2 -3119.384} C_VEL
LIN {X 0,Y 551.946,Z 322.221,A -85,B 0,C 180,E1 -3121.894,E2 -3121.894} C_VEL
LIN {X 0,Y 551.903,Z 327.609,A -85,B 0,C 180,E1 -3125.152,E2 -3125.152} C_VEL
LIN {X 0,Y 551.828,Z 331.656,A -85,B 0,C 180,E1 -3127.539,E2 -3127.539} C_VEL
LIN {X 0,Y 551.818,Z 337.049,A -85,B 0,C 180,E1 -3130.663,E2 -3130.663} C_VEL
LIN {X 0,Y 551.721,Z 342.4,A -85,B 0,C 180,E1 -3133.726,E2 -3133.726} C_VEL
LIN {X 0,Y 551.725,Z 346.547,A -85,B 0,C 180,E1 -3135.994,E2 -3135.994} C_VEL
LIN {X 0,Y 551.709,Z 348.534,A -85,B 0,C 180,E1 -3137.073,E2 -3137.073} C_VEL
LIN {X 0,Y 553.039,Z 357.347,A -85,B 0,C 180,E1 -3137.314,E2 -3137.314} C_VEL
LIN {X 0,Y 552.863,Z 369.824,A -85,B 0,C 180,E1 -3137.707,E2 -3137.707} C_VEL
LIN {X 0,Y 552.667,Z 382.329,A -85,B 0,C 180,E1 -3138.261,E2 -3138.261} C_VEL
LIN {X 0,Y 552.567,Z 393.828,A -85,B 0,C 180,E1 -3138.931,E2 -3138.931} C_VEL
LIN {X 0,Y 552.354,Z 404.866,A -85,B 0,C 180,E1 -3139.74,E2 -3139.74} C_VEL
LIN {X 0,Y 552.175,Z 414.905,A -85,B 0,C 180,E1 -3140.661,E2 -3140.661} C_VEL
LIN {X 0,Y 552.007,Z 424.604,A -85,B 0,C 180,E1 -3141.766,E2 -3141.766} C_VEL
LIN {X 0,Y 551.894,Z 432.463,A -85,B 0,C 180,E1 -3142.887,E2 -3142.887} C_VEL
LIN {X 0,Y 551.868,Z 439.459,A -85,B 0,C 180,E1 -3144.153,E2 -3144.153} C_VEL
LIN {X 0,Y 551.725,Z 444.199,A -85,B 0,C 180,E1 -3145.251,E2 -3145.251} C_VEL
LIN {X 0,Y 551.75,Z 447.831,A -85,B 0,C 180,E1 -3146.349,E2 -3146.349} C_VEL
LIN {X 0,Y 551.723,Z 449.707,A -85,B 0,C 180,E1 -3147.08,E2 -3147.08} C_VEL
LIN {X 0,Y 551.657,Z 451.129,A -85,B 0,C 180,E1 -3147.81,E2 -3147.81} C_VEL
LIN {X 0,Y 551.642,Z 452.758,A -85,B 0,C 180,E1 -3149.27,E2 -3149.27} C_VEL
LIN {X 0,Y 551.641,Z 452.996,A -85,B 0,C 180,E1 -3150,E2 -3150} C_VEL
LIN {X 0,Y 551.641,Z 452.814,A -85,B 0,C 180,E1 -3150.73,E2 -3150.73} C_VEL
LIN {X 0,Y 551.657,Z 451.264,A -85,B 0,C 180,E1 -3152.191,E2 -3152.191} C_VEL
LIN {X 0,Y 551.724,Z 449.903,A -85,B 0,C 180,E1 -3152.921,E2 -3152.921} C_VEL
LIN {X 0,Y 551.764,Z 447.025,A -85,B 0,C 180,E1 -3154.017,E2 -3154.017} C_VEL
LIN {X 0,Y 551.723,Z 443.124,A -85,B 0,C 180,E1 -3155.116,E2 -3155.116} C_VEL
LIN {X 0,Y 551.811,Z 437.391,A -85,B 0,C 180,E1 -3156.35,E2 -3156.35} C_VEL
LIN {X 0,Y 551.925,Z 430.536,A -85,B 0,C 180,E1 -3157.5,E2 -3157.5} C_VEL
LIN {X 0,Y 552.063,Z 422.353,A -85,B 0,C 180,E1 -3158.603,E2 -3158.603} C_VEL
LIN {X 0,Y 552.197,Z 413.985,A -85,B 0,C 180,E1 -3159.524,E2 -3159.524} C_VEL
LIN {X 0,Y 552.403,Z 403.663,A -85,B 0,C 180,E1 -3160.445,E2 -3160.445} C_VEL
LIN {X 0,Y 552.555,Z 392.052,A -85,B 0,C 180,E1 -3161.275,E2 -3161.275} C_VEL
LIN {X 0,Y 552.701,Z 380.443,A -85,B 0,C 180,E1 -3161.925,E2 -3161.925} C_VEL
LIN {X 0,Y 552.925,Z 368.428,A -85,B 0,C 180,E1 -3162.432,E2 -3162.432} C_VEL
LIN {X 0,Y 552.865,Z 355.367,A -85,B 0,C 180,E1 -3162.83,E2 -3162.83} C_VEL
LIN {X 0,Y 551.685,Z 348.527,A -85,B 0,C 180,E1 -3163.022,E2 -3163.022} C_VEL
LIN {X 0,Y 551.736,Z 343.945,A -85,B 0,C 180,E1 -3165.515,E2 -3165.515} C_VEL
LIN {X 0,Y 551.715,Z 339.878,A -85,B 0,C 180,E1 -3167.802,E2 -3167.802} C_VEL
LIN {X 0,Y 551.775,Z 335.887,A -85,B 0,C 180,E1 -3170.115,E2 -3170.115} C_VEL
LIN {X 0,Y 551.829,Z 331.808,A -85,B 0,C 180,E1 -3172.462,E2 -3172.462} C_VEL
LIN {X 0,Y 551.904,Z 327.014,A -85,B 0,C 180,E1 -3175.294,E2 -3175.294} C_VEL
LIN {X 0,Y 551.987,Z 321.666,A -85,B 0,C 180,E1 -3178.535,E2 -3178.535} C_VEL
LIN {X 0,Y 552.028,Z 316.958,A -85,B 0,C 180,E1 -3181.465,E2 -3181.465} C_VEL
LIN {X 0,Y 552.088,Z 312.676,A -85,B 0,C 180,E1 -3184.163,E2 -3184.163} C_VEL
LIN {X 0,Y 552.025,Z 310.725,A -85,B 0,C 180,E1 -3185.432,E2 -3185.432} C_VEL
LIN {X 0,Y 552.092,Z 310.712,A -85,B 0,C 180,E1 -3187.885,E2 -3187.885} C_VEL
LIN {X 0,Y 552.11,Z 310.714,A -85,B 0,C 180,E1 -3190.481,E2 -3190.481} C_VEL
LIN {X 0,Y 552.102,Z 310.713,A -85,B 0,C 180,E1 -3193.482,E2 -3193.482} C_VEL
LIN {X 0,Y 552.07,Z 310.714,A -85,B 0,C 180,E1 -3196.572,E2 -3196.572} C_VEL
LIN {X 0,Y 552.106,Z 310.71,A -85,B 0,C 180,E1 -3199.797,E2 -3199.797} C_VEL
LIN {X 0,Y 552.088,Z 310.717,A -85,B 0,C 180,E1 -3202.336,E2 -3202.336} C_VEL
LIN {X 0,Y 552.118,Z 310.709,A -85,B 0,C 180,E1 -3205.053,E2 -3205.053} C_VEL
LIN {X 0,Y 552.125,Z 310.711,A -85,B 0,C 180,E1 -3207.682,E2 -3207.682} C_VEL
LIN {X 0,Y 552.082,Z 310.712,A -85,B 0,C 180,E1 -3210.233,E2 -3210.233} C_VEL
LIN {X 0,Y 552.087,Z 310.715,A -85,B 0,C 180,E1 -3213.009,E2 -3213.009} C_VEL
LIN {X 0,Y 552.084,Z 310.718,A -85,B 0,C 180,E1 -3215.961,E2 -3215.961} C_VEL
LIN {X 0,Y 552.123,Z 310.711,A -85,B 0,C 180,E1 -3219.12,E2 -3219.12} C_VEL
LIN {X 0,Y 552.119,Z 310.712,A -85,B 0,C 180,E1 -3221.444,E2 -3221.444} C_VEL
LIN {X 0,Y 552.102,Z 310.709,A -85,B 0,C 180,E1 -3223.737,E2 -3223.737} C_VEL
LIN {X 0,Y 552.108,Z 310.712,A -85,B 0,C 180,E1 -3226.004,E2 -3226.004} C_VEL
LIN {X 0,Y 552.156,Z 310.704,A -85,B 0,C 180,E1 -3228.993,E2 -3228.993} C_VEL
LIN {X 0,Y 552.155,Z 310.706,A -85,B 0,C 180,E1 -3231.951,E2 -3231.951} C_VEL
LIN {X 0,Y 552.226,Z 310.701,A -85,B 0,C 180,E1 -3234.889,E2 -3234.889} C_VEL
LIN {X 0,Y 552.22,Z 310.696,A -85,B 0,C 180,E1 -3237.812,E2 -3237.812} C_VEL
LIN {X 0,Y 552.221,Z 310.696,A -85,B 0,C 180,E1 -3240.729,E2 -3240.729} C_VEL
LIN {X 0,Y 552.191,Z 310.701,A -85,B 0,C 180,E1 -3242.918,E2 -3242.918} C_VEL
LIN {X 0,Y 552.208,Z 310.698,A -85,B 0,C 180,E1 -3245.844,E2 -3245.844} C_VEL
LIN {X 0,Y 552.165,Z 310.707,A -85,B 0,C 180,E1 -3248.786,E2 -3248.786} C_VEL
LIN {X 0,Y 552.153,Z 310.707,A -85,B 0,C 180,E1 -3251.751,E2 -3251.751} C_VEL
LIN {X 0,Y 552.115,Z 310.709,A -85,B 0,C 180,E1 -3254.749,E2 -3254.749} C_VEL
LIN {X 0,Y 552.104,Z 310.711,A -85,B 0,C 180,E1 -3257.789,E2 -3257.789} C_VEL
LIN {X 0,Y 552.129,Z 310.709,A -85,B 0,C 180,E1 -3260.101,E2 -3260.101} C_VEL
LIN {X 0,Y 552.092,Z 310.716,A -85,B 0,C 180,E1 -3262.451,E2 -3262.451} C_VEL
LIN {X 0,Y 552.131,Z 310.709,A -85,B 0,C 180,E1 -3265.346,E2 -3265.346} C_VEL
LIN {X 0,Y 552.05,Z 310.717,A -85,B 0,C 180,E1 -3268.102,E2 -3268.102} C_VEL
LIN {X 0,Y 552.093,Z 310.715,A -85,B 0,C 180,E1 -3270.61,E2 -3270.61} C_VEL
LIN {X 0,Y 552.118,Z 310.71,A -85,B 0,C 180,E1 -3273.186,E2 -3273.186} C_VEL
LIN {X 0,Y 552.106,Z 310.715,A -85,B 0,C 180,E1 -3275.842,E2 -3275.842} C_VEL
LIN {X 0,Y 552.115,Z 310.711,A -85,B 0,C 180,E1 -3279.061,E2 -3279.061} C_VEL
LIN {X 0,Y 552.07,Z 310.717,A -85,B 0,C 180,E1 -3281.451,E2 -3281.451} C_VEL
LIN {X 0,Y 552.075,Z 310.72,A -85,B 0,C 180,E1 -3284.53,E2 -3284.53} C_VEL
LIN {X 0,Y 552.13,Z 310.71,A -85,B 0,C 180,E1 -3287.585,E2 -3287.585} C_VEL
LIN {X 0,Y 552.128,Z 310.709,A -85,B 0,C 180,E1 -3290.473,E2 -3290.473} C_VEL
LIN {X 0,Y 552.131,Z 310.814,A -85,B 0,C 180,E1 -3293.141,E2 -3293.141} C_VEL
LIN {X 0,Y 552.542,Z 314.102,A -85,B 0,C 180,E1 -3294.493,E2 -3294.493} C_VEL
LIN {X 0,Y 552.509,Z 320.713,A -85,B 0,C 180,E1 -3297.091,E2 -3297.091} C_VEL
LIN {X 0,Y 552.383,Z 328.054,A -85,B 0,C 180,E1 -3299.902,E2 -3299.902} C_VEL
LIN {X 0,Y 552.267,Z 336.31,A -85,B 0,C 180,E1 -3302.974,E2 -3302.974} C_VEL
LIN {X 0,Y 552.159,Z 344.561,A -85,B 0,C 180,E1 -3305.965,E2 -3305.965} C_VEL
LIN {X 0,Y 552.07,Z 352.352,A -85,B 0,C 180,E1 -3308.727,E2 -3308.727} C_VEL
LIN {X 0,Y 551.952,Z 360.144,A -85,B 0,C 180,E1 -3311.438,E2 -3311.438} C_VEL
LIN {X 0,Y 551.903,Z 369.048,A -85,B 0,C 180,E1 -3314.489,E2 -3314.489} C_VEL
LIN {X 0,Y 551.837,Z 376.491,A -85,B 0,C 180,E1 -3317.005,E2 -3317.005} C_VEL
LIN {X 0,Y 553.086,Z 385.435,A -85,B 0,C 180,E1 -3317.222,E2 -3317.222} C_VEL
LIN {X 0,Y 552.934,Z 398.471,A -85,B 0,C 180,E1 -3317.614,E2 -3317.614} C_VEL
LIN {X 0,Y 552.741,Z 409.483,A -85,B 0,C 180,E1 -3318.076,E2 -3318.076} C_VEL
LIN {X 0,Y 552.577,Z 421.229,A -85,B 0,C 180,E1 -3318.717,E2 -3318.717} C_VEL
LIN {X 0,Y 552.43,Z 431.926,A -85,B 0,C 180,E1 -3319.462,E2 -3319.462} C_VEL
LIN {X 0,Y 552.233,Z 441.6,A -85,B 0,C 180,E1 -3320.292,E2 -3320.292} C_VEL
LIN {X 0,Y 552.079,Z 450.412,A -85,B 0,C 180,E1 -3321.213,E2 -3321.213} C_VEL
LIN {X 0,Y 551.95,Z 458.999,A -85,B 0,C 180,E1 -3322.317,E2 -3322.317} C_VEL
LIN {X 0,Y 551.823,Z 465.866,A -85,B 0,C 180,E1 -3323.418,E2 -3323.418} C_VEL
LIN {X 0,Y 551.804,Z 471.365,A -85,B 0,C 180,E1 -3324.518,E2 -3324.518} C_VEL
LIN {X 0,Y 551.764,Z 475.677,A -85,B 0,C 180,E1 -3325.617,E2 -3325.617} C_VEL
LIN {X 0,Y 551.75,Z 477.956,A -85,B 0,C 180,E1 -3326.348,E2 -3326.348} C_VEL
LIN {X 0,Y 551.723,Z 479.808,A -85,B 0,C 180,E1 -3327.079,E2 -3327.079} C_VEL
LIN {X 0,Y 551.657,Z 481.199,A -85,B 0,C 180,E1 -3327.809,E2 -3327.809} C_VEL
LIN {X 0,Y 551.641,Z 482.784,A -85,B 0,C 180,E1 -3329.27,E2 -3329.27} C_VEL
LIN {X 0,Y 551.64,Z 483,A -85,B 0,C 180,E1 -3330,E2 -3330} C_VEL
LIN {X 0,Y 551.645,Z 482.186,A -85,B 0,C 180,E1 -3331.46,E2 -3331.46} C_VEL
LIN {X 0,Y 551.657,Z 481.201,A -85,B 0,C 180,E1 -3332.19,E2 -3332.19} C_VEL
LIN {X 0,Y 551.723,Z 479.811,A -85,B 0,C 180,E1 -3332.92,E2 -3332.92} C_VEL
LIN {X 0,Y 551.764,Z 476.897,A -85,B 0,C 180,E1 -3334.017,E2 -3334.017} C_VEL
LIN {X 0,Y 551.723,Z 472.951,A -85,B 0,C 180,E1 -3335.115,E2 -3335.115} C_VEL
LIN {X 0,Y 551.822,Z 467.205,A -85,B 0,C 180,E1 -3336.339,E2 -3336.339} C_VEL
LIN {X 0,Y 551.926,Z 460.24,A -85,B 0,C 180,E1 -3337.499,E2 -3337.499} C_VEL
LIN {X 0,Y 552.082,Z 451.994,A -85,B 0,C 180,E1 -3338.602,E2 -3338.602} C_VEL
LIN {X 0,Y 552.2,Z 443.543,A -85,B 0,C 180,E1 -3339.523,E2 -3339.523} C_VEL
LIN {X 0,Y 552.422,Z 433.103,A -85,B 0,C 180,E1 -3340.444,E2 -3340.444} C_VEL
LIN {X 0,Y 552.577,Z 421.359,A -85,B 0,C 180,E1 -3341.275,E2 -3341.275} C_VEL
LIN {X 0,Y 552.745,Z 409.496,A -85,B 0,C 180,E1 -3341.923,E2 -3341.923} C_VEL
LIN {X 0,Y 552.955,Z 397.189,A -85,B 0,C 180,E1 -3342.431,E2 -3342.431} C_VEL
LIN {X 0,Y 553.064,Z 384.064,A -85,B 0,C 180,E1 -3342.813,E2 -3342.813} C_VEL
LIN {X 0,Y 551.837,Z 376.493,A -85,B 0,C 180,E1 -3342.994,E2 -3342.994} C_VEL
LIN {X 0,Y 551.901,Z 367.937,A -85,B 0,C 180,E1 -3345.889,E2 -3345.889} C_VEL
LIN {X 0,Y 551.994,Z 359.033,A -85,B 0,C 180,E1 -3348.945,E2 -3348.945} C_VEL
LIN {X 0,Y 552.077,Z 351.213,A -85,B 0,C 180,E1 -3351.674,E2 -3351.674} C_VEL
LIN {X 0,Y 552.178,Z 343.45,A -85,B 0,C 180,E1 -3354.434,E2 -3354.434} C_VEL
LIN {X 0,Y 552.291,Z 335.659,A -85,B 0,C 180,E1 -3357.264,E2 -3357.264} C_VEL
LIN {X 0,Y 552.381,Z 328.056,A -85,B 0,C 180,E1 -3360.097,E2 -3360.097} C_VEL
LIN {X 0,Y 552.506,Z 320.715,A -85,B 0,C 180,E1 -3362.909,E2 -3362.909} C_VEL
LIN {X 0,Y 552.58,Z 314.095,A -85,B 0,C 180,E1 -3365.513,E2 -3365.513} C_VEL
LIN {X 0,Y 552.126,Z 310.714,A -85,B 0,C 180,E1 -3366.972,E2 -3366.972} C_VEL
LIN {X 0,Y 552.13,Z 310.709,A -85,B 0,C 180,E1 -3369.526,E2 -3369.526} C_VEL
LIN {X 0,Y 552.126,Z 310.711,A -85,B 0,C 180,E1 -3372.424,E2 -3372.424} C_VEL
LIN {X 0,Y 552.092,Z 310.717,A -85,B 0,C 180,E1 -3375.562,E2 -3375.562} C_VEL
LIN {X 0,Y 552.067,Z 310.717,A -85,B 0,C 180,E1 -3378.549,E2 -3378.549} C_VEL
LIN {X 0,Y 552.11,Z 310.709,A -85,B 0,C 180,E1 -3381.41,E2 -3381.41} C_VEL
LIN {X 0,Y 552.106,Z 310.716,A -85,B 0,C 180,E1 -3384.158,E2 -3384.158} C_VEL
LIN {X 0,Y 552.115,Z 310.71,A -85,B 0,C 180,E1 -3386.814,E2 -3386.814} C_VEL
LIN {X 0,Y 552.089,Z 310.716,A -85,B 0,C 180,E1 -3389.39,E2 -3389.39} C_VEL
LIN {X 0,Y 552.046,Z 310.717,A -85,B 0,C 180,E1 -3391.898,E2 -3391.898} C_VEL
LIN {X 0,Y 552.127,Z 310.709,A -85,B 0,C 180,E1 -3394.653,E2 -3394.653} C_VEL
LIN {X 0,Y 552.088,Z 310.717,A -85,B 0,C 180,E1 -3397.549,E2 -3397.549} C_VEL
LIN {X 0,Y 552.14,Z 310.706,A -85,B 0,C 180,E1 -3400.373,E2 -3400.373} C_VEL
LIN {X 0,Y 552.122,Z 310.713,A -85,B 0,C 180,E1 -3402.976,E2 -3402.976} C_VEL
LIN {X 0,Y 552.113,Z 310.712,A -85,B 0,C 180,E1 -3406.004,E2 -3406.004} C_VEL
LIN {X 0,Y 552.151,Z 310.704,A -85,B 0,C 180,E1 -3408.993,E2 -3408.993} C_VEL
LIN {X 0,Y 552.155,Z 310.705,A -85,B 0,C 180,E1 -3411.951,E2 -3411.951} C_VEL
LIN {X 0,Y 552.223,Z 310.701,A -85,B 0,C 180,E1 -3414.889,E2 -3414.889} C_VEL
LIN {X 0,Y 552.217,Z 310.698,A -85,B 0,C 180,E1 -3417.812,E2 -3417.812} C_VEL
LIN {X 0,Y 552.217,Z 310.696,A -85,B 0,C 180,E1 -3420.729,E2 -3420.729} C_VEL
LIN {X 0,Y 552.189,Z 310.7,A -85,B 0,C 180,E1 -3422.918,E2 -3422.918} C_VEL
LIN {X 0,Y 552.205,Z 310.698,A -85,B 0,C 180,E1 -3425.844,E2 -3425.844} C_VEL
LIN {X 0,Y 552.161,Z 310.708,A -85,B 0,C 180,E1 -3428.786,E2 -3428.786} C_VEL
LIN {X 0,Y 552.149,Z 310.709,A -85,B 0,C 180,E1 -3431.751,E2 -3431.751} C_VEL
LIN {X 0,Y 552.116,Z 310.708,A -85,B 0,C 180,E1 -3434.749,E2 -3434.749} C_VEL
LIN {X 0,Y 552.104,Z 310.71,A -85,B 0,C 180,E1 -3437.789,E2 -3437.789} C_VEL
LIN {X 0,Y 552.125,Z 310.709,A -85,B 0,C 180,E1 -3440.102,E2 -3440.102} C_VEL
LIN {X 0,Y 552.088,Z 310.718,A -85,B 0,C 180,E1 -3442.451,E2 -3442.451} C_VEL
LIN {X 0,Y 552.127,Z 310.71,A -85,B 0,C 180,E1 -3445.347,E2 -3445.347} C_VEL
LIN {X 0,Y 552.046,Z 310.717,A -85,B 0,C 180,E1 -3448.102,E2 -3448.102} C_VEL
LIN {X 0,Y 552.088,Z 310.715,A -85,B 0,C 180,E1 -3450.622,E2 -3450.622} C_VEL
LIN {X 0,Y 552.116,Z 310.709,A -85,B 0,C 180,E1 -3453.186,E2 -3453.186} C_VEL
LIN {X 0,Y 552.108,Z 310.711,A -85,B 0,C 180,E1 -3453.801,E2 -3453.801} C_VEL
LIN {X 0,Y 551.473,Z 310.794,A -85,B 0,C 180,E1 -3454.41,E2 -3454.41} C_VEL
LIN {X 0,Y 548.651,Z 311.144,A -85,B 0,C 180,E1 -3455.398,E2 -3455.398} C_VEL
LIN {X 0,Y 546.23,Z 311.447,A -85,B 0,C 180,E1 -3456.193,E2 -3456.193} C_VEL
LIN {X 0,Y 545.16,Z 311.576,A -85,B 0,C 180,E1 -3456.807,E2 -3456.807} C_VEL
LIN {X 0,Y 545.058,Z 311.589,A -85,B 0,C 180,E1 -3457.015,E2 -3457.015} C_VEL
LIN {X 0,Y 545.058,Z 311.588,A -85,B 0,C 180,E1 -3460.144,E2 -3460.144} C_VEL
LIN {X 0,Y 545.016,Z 311.596,A -85,B 0,C 180,E1 -3463.113,E2 -3463.113} C_VEL
LIN {X 0,Y 545.052,Z 311.594,A -85,B 0,C 180,E1 -3466.226,E2 -3466.226} C_VEL
LIN {X 0,Y 545.098,Z 311.583,A -85,B 0,C 180,E1 -3468.888,E2 -3468.888} C_VEL
LIN {X 0,Y 545.049,Z 311.592,A -85,B 0,C 180,E1 -3471.764,E2 -3471.764} C_VEL
LIN {X 0,Y 544.988,Z 311.599,A -85,B 0,C 180,E1 -3474.334,E2 -3474.334} C_VEL
LIN {X 0,Y 544.983,Z 311.601,A -85,B 0,C 180,E1 -3474.529,E2 -3474.529} C_VEL
LIN {X 0,Y 545.019,Z 314.154,A -85,B 0,C 180,E1 -3476.326,E2 -3476.326} C_VEL
LIN {X 0,Y 544.952,Z 318.264,A -85,B 0,C 180,E1 -3478.946,E2 -3478.946} C_VEL
LIN {X 0,Y 544.935,Z 322.329,A -85,B 0,C 180,E1 -3481.499,E2 -3481.499} C_VEL
LIN {X 0,Y 544.857,Z 327.741,A -85,B 0,C 180,E1 -3484.808,E2 -3484.808} C_VEL
LIN {X 0,Y 544.78,Z 331.787,A -85,B 0,C 180,E1 -3487.232,E2 -3487.232} C_VEL
LIN {X 0,Y 544.734,Z 337.213,A -85,B 0,C 180,E1 -3490.401,E2 -3490.401} C_VEL
LIN {X 0,Y 544.646,Z 342.546,A -85,B 0,C 180,E1 -3493.509,E2 -3493.509} C_VEL
LIN {X 0,Y 544.662,Z 346.567,A -85,B 0,C 180,E1 -3495.809,E2 -3495.809} C_VEL
LIN {X 0,Y 544.602,Z 348.536,A -85,B 0,C 180,E1 -3496.901,E2 -3496.901} C_VEL
LIN {X 0,Y 546.109,Z 358.283,A -85,B 0,C 180,E1 -3497.174,E2 -3497.174} C_VEL
LIN {X 0,Y 545.917,Z 371.039,A -85,B 0,C 180,E1 -3497.595,E2 -3497.595} C_VEL
LIN {X 0,Y 545.693,Z 383.757,A -85,B 0,C 180,E1 -3498.184,E2 -3498.184} C_VEL
LIN {X 0,Y 545.559,Z 394.925,A -85,B 0,C 180,E1 -3498.859,E2 -3498.859} C_VEL
LIN {X 0,Y 545.34,Z 405.96,A -85,B 0,C 180,E1 -3499.7,E2 -3499.7} C_VEL
LIN {X 0,Y 545.122,Z 416.691,A -85,B 0,C 180,E1 -3500.726,E2 -3500.726} C_VEL
LIN {X 0,Y 544.975,Z 424.608,A -85,B 0,C 180,E1 -3501.659,E2 -3501.659} C_VEL
LIN {X 0,Y 544.829,Z 432.355,A -85,B 0,C 180,E1 -3502.775,E2 -3502.775} C_VEL
LIN {X 0,Y 544.778,Z 439.462,A -85,B 0,C 180,E1 -3504.077,E2 -3504.077} C_VEL
LIN {X 0,Y 544.628,Z 444.201,A -85,B 0,C 180,E1 -3505.189,E2 -3505.189} C_VEL
LIN {X 0,Y 544.669,Z 447.832,A -85,B 0,C 180,E1 -3506.301,E2 -3506.301} C_VEL
LIN {X 0,Y 544.65,Z 449.709,A -85,B 0,C 180,E1 -3507.042,E2 -3507.042} C_VEL
LIN {X 0,Y 544.572,Z 451.129,A -85,B 0,C 180,E1 -3507.782,E2 -3507.782} C_VEL
LIN {X 0,Y 544.542,Z 452.757,A -85,B 0,C 180,E1 -3509.261,E2 -3509.261} C_VEL
LIN {X 0,Y 544.542,Z 452.996,A -85,B 0,C 180,E1 -3510,E2 -3510} C_VEL
LIN {X 0,Y 544.542,Z 452.814,A -85,B 0,C 180,E1 -3510.74,E2 -3510.74} C_VEL
LIN {X 0,Y 544.572,Z 451.262,A -85,B 0,C 180,E1 -3512.219,E2 -3512.219} C_VEL
LIN {X 0,Y 544.651,Z 449.901,A -85,B 0,C 180,E1 -3512.959,E2 -3512.959} C_VEL
LIN {X 0,Y 544.684,Z 447.023,A -85,B 0,C 180,E1 -3514.07,E2 -3514.07} C_VEL
LIN {X 0,Y 544.653,Z 443.121,A -85,B 0,C 180,E1 -3515.183,E2 -3515.183} C_VEL
LIN {X 0,Y 544.725,Z 437.895,A -85,B 0,C 180,E1 -3516.336,E2 -3516.336} C_VEL
LIN {X 0,Y 544.859,Z 430.531,A -85,B 0,C 180,E1 -3517.598,E2 -3517.598} C_VEL
LIN {X 0,Y 544.999,Z 422.349,A -85,B 0,C 180,E1 -3518.715,E2 -3518.715} C_VEL
LIN {X 0,Y 545.16,Z 413.978,A -85,B 0,C 180,E1 -3519.648,E2 -3519.648} C_VEL
LIN {X 0,Y 545.405,Z 403.653,A -85,B 0,C 180,E1 -3520.581,E2 -3520.581} C_VEL
LIN {X 0,Y 545.558,Z 392.449,A -85,B 0,C 180,E1 -3521.394,E2 -3521.394} C_VEL
LIN {X 0,Y 545.712,Z 382.247,A -85,B 0,C 180,E1 -3521.986,E2 -3521.986} C_VEL
LIN {X 0,Y 545.979,Z 369.711,A -85,B 0,C 180,E1 -3522.546,E2 -3522.546} C_VEL
LIN {X 0,Y 546.02,Z 356.717,A -85,B 0,C 180,E1 -3522.958,E2 -3522.958} C_VEL
LIN {X 0,Y 544.611,Z 348.525,A -85,B 0,C 180,E1 -3523.194,E2 -3523.194} C_VEL
LIN {X 0,Y 544.639,Z 344.052,A -85,B 0,C 180,E1 -3525.723,E2 -3525.723} C_VEL
LIN {X 0,Y 544.645,Z 340.056,A -85,B 0,C 180,E1 -3528.041,E2 -3528.041} C_VEL
LIN {X 0,Y 544.708,Z 336.003,A -85,B 0,C 180,E1 -3530.387,E2 -3530.387} C_VEL
LIN {X 0,Y 544.782,Z 331.938,A -85,B 0,C 180,E1 -3532.769,E2 -3532.769} C_VEL
LIN {X 0,Y 544.834,Z 327.463,A -85,B 0,C 180,E1 -3535.45,E2 -3535.45} C_VEL
LIN {X 0,Y 544.923,Z 322.131,A -85,B 0,C 180,E1 -3538.715,E2 -3538.715} C_VEL
LIN {X 0,Y 544.97,Z 317.048,A -85,B 0,C 180,E1 -3541.92,E2 -3541.92} C_VEL
LIN {X 0,Y 545.034,Z 312.897,A -85,B 0,C 180,E1 -3544.566,E2 -3544.566} C_VEL
LIN {X 0,Y 544.99,Z 311.6,A -85,B 0,C 180,E1 -3545.472,E2 -3545.472} C_VEL
LIN {X 0,Y 545.045,Z 311.591,A -85,B 0,C 180,E1 -3548.135,E2 -3548.135} C_VEL
LIN {X 0,Y 545.082,Z 311.59,A -85,B 0,C 180,E1 -3550.472,E2 -3550.472} C_VEL
LIN {X 0,Y 545.079,Z 311.585,A -85,B 0,C 180,E1 -3553.106,E2 -3553.106} C_VEL
LIN {X 0,Y 545.045,Z 311.589,A -85,B 0,C 180,E1 -3556.226,E2 -3556.226} C_VEL
LIN {X 0,Y 545.025,Z 311.597,A -85,B 0,C 180,E1 -3558.88,E2 -3558.88} C_VEL
LIN {X 0,Y 545.046,Z 311.591,A -85,B 0,C 180,E1 -3561.762,E2 -3561.762} C_VEL
LIN {X 0,Y 545.055,Z 311.59,A -85,B 0,C 180,E1 -3564.533,E2 -3564.533} C_VEL
LIN {X 0,Y 545.079,Z 311.588,A -85,B 0,C 180,E1 -3567.212,E2 -3567.212} C_VEL
LIN {X 0,Y 545.057,Z 311.588,A -85,B 0,C 180,E1 -3569.81,E2 -3569.81} C_VEL
LIN {X 0,Y 545.03,Z 311.596,A -85,B 0,C 180,E1 -3572.838,E2 -3572.838} C_VEL
LIN {X 0,Y 545.023,Z 311.594,A -85,B 0,C 180,E1 -3575.629,E2 -3575.629} C_VEL
LIN {X 0,Y 545.059,Z 311.59,A -85,B 0,C 180,E1 -3578.18,E2 -3578.18} C_VEL
LIN {X 0,Y 545.114,Z 311.581,A -85,B 0,C 180,E1 -3580.415,E2 -3580.415} C_VEL
LIN {X 0,Y 545.06,Z 311.587,A -85,B 0,C 180,E1 -3583.521,E2 -3583.521} C_VEL
LIN {X 0,Y 545.073,Z 311.587,A -85,B 0,C 180,E1 -3585.819,E2 -3585.819} C_VEL
LIN {X 0,Y 545.112,Z 311.582,A -85,B 0,C 180,E1 -3588.849,E2 -3588.849} C_VEL
LIN {X 0,Y 545.125,Z 311.583,A -85,B 0,C 180,E1 -3591.847,E2 -3591.847} C_VEL
LIN {X 0,Y 545.202,Z 311.576,A -85,B 0,C 180,E1 -3594.823,E2 -3594.823} C_VEL
LIN {X 0,Y 545.191,Z 311.571,A -85,B 0,C 180,E1 -3597.784,E2 -3597.784} C_VEL
LIN {X 0,Y 545.193,Z 311.571,A -85,B 0,C 180,E1 -3600.739,E2 -3600.739} C_VEL
LIN {X 0,Y 545.159,Z 311.577,A -85,B 0,C 180,E1 -3602.956,E2 -3602.956} C_VEL
LIN {X 0,Y 545.179,Z 311.574,A -85,B 0,C 180,E1 -3605.919,E2 -3605.919} C_VEL
LIN {X 0,Y 545.122,Z 311.583,A -85,B 0,C 180,E1 -3608.9,E2 -3608.9} C_VEL
LIN {X 0,Y 545.096,Z 311.588,A -85,B 0,C 180,E1 -3611.905,E2 -3611.905} C_VEL
LIN {X 0,Y 545.071,Z 311.587,A -85,B 0,C 180,E1 -3614.944,E2 -3614.944} C_VEL
LIN {X 0,Y 545.072,Z 311.587,A -85,B 0,C 180,E1 -3618.026,E2 -3618.026} C_VEL
LIN {X 0,Y 545.094,Z 311.588,A -85,B 0,C 180,E1 -3620.372,E2 -3620.372} C_VEL
LIN {X 0,Y 545.087,Z 311.586,A -85,B 0,C 180,E1 -3623.559,E2 -3623.559} C_VEL
LIN {X 0,Y 545.058,Z 311.59,A -85,B 0,C 180,E1 -3626.002,E2 -3626.002} C_VEL
LIN {X 0,Y 545.039,Z 311.592,A -85,B 0,C 180,E1 -3628.74,E2 -3628.74} C_VEL
LIN {X 0,Y 545.055,Z 311.589,A -85,B 0,C 180,E1 -3631.679,E2 -3631.679} C_VEL
LIN {X 0,Y 545.074,Z 311.59,A -85,B 0,C 180,E1 -3634.564,E2 -3634.564} C_VEL
LIN {X 0,Y 545.035,Z 311.593,A -85,B 0,C 180,E1 -3637.304,E2 -3637.304} C_VEL
LIN {X 0,Y 545.06,Z 311.587,A -85,B 0,C 180,E1 -3640.143,E2 -3640.143} C_VEL
LIN {X 0,Y 545.014,Z 311.597,A -85,B 0,C 180,E1 -3643.113,E2 -3643.113} C_VEL
LIN {X 0,Y 545.048,Z 311.596,A -85,B 0,C 180,E1 -3646.227,E2 -3646.227} C_VEL
LIN {X 0,Y 545.087,Z 311.585,A -85,B 0,C 180,E1 -3648.886,E2 -3648.886} C_VEL
LIN {X 0,Y 545.048,Z 311.595,A -85,B 0,C 180,E1 -3651.763,E2 -3651.763} C_VEL
LIN {X 0,Y 545.12,Z 311.76,A -85,B 0,C 180,E1 -3652.996,E2 -3652.996} C_VEL
LIN {X 0,Y 545.602,Z 316.68,A -85,B 0,C 180,E1 -3655.026,E2 -3655.026} C_VEL
LIN {X 0,Y 545.473,Z 323.414,A -85,B 0,C 180,E1 -3657.677,E2 -3657.677} C_VEL
LIN {X 0,Y 545.344,Z 331.205,A -85,B 0,C 180,E1 -3660.678,E2 -3660.678} C_VEL
LIN {X 0,Y 545.199,Z 338.996,A -85,B 0,C 180,E1 -3663.594,E2 -3663.594} C_VEL
LIN {X 0,Y 545.103,Z 346.787,A -85,B 0,C 180,E1 -3666.442,E2 -3666.442} C_VEL
LIN {X 0,Y 544.991,Z 354.579,A -85,B 0,C 180,E1 -3669.229,E2 -3669.229} C_VEL
LIN {X 0,Y 544.883,Z 362.37,A -85,B 0,C 180,E1 -3671.968,E2 -3671.968} C_VEL
LIN {X 0,Y 544.817,Z 370.161,A -85,B 0,C 180,E1 -3674.666,E2 -3674.666} C_VEL
LIN {X 0,Y 544.756,Z 376.491,A -85,B 0,C 180,E1 -3676.833,E2 -3676.833} C_VEL
LIN {X 0,Y 546.166,Z 386.35,A -85,B 0,C 180,E1 -3677.081,E2 -3677.081} C_VEL
LIN {X 0,Y 545.975,Z 399.766,A -85,B 0,C 180,E1 -3677.501,E2 -3677.501} C_VEL
LIN {X 0,Y 545.777,Z 411.41,A -85,B 0,C 180,E1 -3678.016,E2 -3678.016} C_VEL
LIN {X 0,Y 545.556,Z 423.608,A -85,B 0,C 180,E1 -3678.727,E2 -3678.727} C_VEL
LIN {X 0,Y 545.418,Z 434.257,A -85,B 0,C 180,E1 -3679.513,E2 -3679.513} C_VEL
LIN {X 0,Y 545.165,Z 443.537,A -85,B 0,C 180,E1 -3680.352,E2 -3680.352} C_VEL
LIN {X 0,Y 545.029,Z 451.989,A -85,B 0,C 180,E1 -3681.285,E2 -3681.285} C_VEL
LIN {X 0,Y 544.86,Z 460.236,A -85,B 0,C 180,E1 -3682.402,E2 -3682.402} C_VEL
LIN {X 0,Y 544.734,Z 467.615,A -85,B 0,C 180,E1 -3683.655,E2 -3683.655} C_VEL
LIN {X 0,Y 544.653,Z 472.949,A -85,B 0,C 180,E1 -3684.817,E2 -3684.817} C_VEL
LIN {X 0,Y 544.684,Z 476.895,A -85,B 0,C 180,E1 -3685.93,E2 -3685.93} C_VEL
LIN {X 0,Y 544.65,Z 479.808,A -85,B 0,C 180,E1 -3687.041,E2 -3687.041} C_VEL
LIN {X 0,Y 544.546,Z 482.185,A -85,B 0,C 180,E1 -3688.521,E2 -3688.521} C_VEL
LIN {X 0,Y 544.541,Z 483,A -85,B 0,C 180,E1 -3690,E2 -3690} C_VEL
LIN {X 0,Y 544.546,Z 482.186,A -85,B 0,C 180,E1 -3691.479,E2 -3691.479} C_VEL
LIN {X 0,Y 544.65,Z 479.811,A -85,B 0,C 180,E1 -3692.958,E2 -3692.958} C_VEL
LIN {X 0,Y 544.684,Z 476.897,A -85,B 0,C 180,E1 -3694.069,E2 -3694.069} C_VEL
LIN {X 0,Y 544.653,Z 472.951,A -85,B 0,C 180,E1 -3695.182,E2 -3695.182} C_VEL
LIN {X 0,Y 544.734,Z 467.613,A -85,B 0,C 180,E1 -3696.346,E2 -3696.346} C_VEL
LIN {X 0,Y 544.859,Z 460.241,A -85,B 0,C 180,E1 -3697.597,E2 -3697.597} C_VEL
LIN {X 0,Y 545.028,Z 451.994,A -85,B 0,C 180,E1 -3698.714,E2 -3698.714} C_VEL
LIN {X 0,Y 545.164,Z 443.543,A -85,B 0,C 180,E1 -3699.647,E2 -3699.647} C_VEL
LIN {X 0,Y 545.419,Z 433.104,A -85,B 0,C 180,E1 -3700.58,E2 -3700.58} C_VEL
LIN {X 0,Y 545.604,Z 421.673,A -85,B 0,C 180,E1 -3701.4,E2 -3701.4} C_VEL
LIN {X 0,Y 545.762,Z 411.422,A -85,B 0,C 180,E1 -3701.984,E2 -3701.984} C_VEL
LIN {X 0,Y 545.974,Z 399.779,A -85,B 0,C 180,E1 -3702.498,E2 -3702.498} C_VEL
LIN {X 0,Y 546.165,Z 386.371,A -85,B 0,C 180,E1 -3702.919,E2 -3702.919} C_VEL
LIN {X 0,Y 544.757,Z 376.493,A -85,B 0,C 180,E1 -3703.166,E2 -3703.166} C_VEL
LIN {X 0,Y 544.844,Z 369.05,A -85,B 0,C 180,E1 -3705.716,E2 -3705.716} C_VEL
LIN {X 0,Y 544.908,Z 360.146,A -85,B 0,C 180,E1 -3708.81,E2 -3708.81} C_VEL
LIN {X 0,Y 545.003,Z 353.467,A -85,B 0,C 180,E1 -3711.165,E2 -3711.165} C_VEL
LIN {X 0,Y 545.141,Z 344.563,A -85,B 0,C 180,E1 -3714.364,E2 -3714.364} C_VEL
LIN {X 0,Y 545.276,Z 336.821,A -85,B 0,C 180,E1 -3717.21,E2 -3717.21} C_VEL
LIN {X 0,Y 545.39,Z 328.633,A -85,B 0,C 180,E1 -3720.302,E2 -3720.302} C_VEL
LIN {X 0,Y 545.51,Z 321.348,A -85,B 0,C 180,E1 -3723.131,E2 -3723.131} C_VEL
LIN {X 0,Y 545.597,Z 315.559,A -85,B 0,C 180,E1 -3725.425,E2 -3725.425} C_VEL
LIN {X 0,Y 545.079,Z 311.592,A -85,B 0,C 180,E1 -3727.135,E2 -3727.135} C_VEL
LIN {X 0,Y 545.088,Z 311.59,A -85,B 0,C 180,E1 -3730.139,E2 -3730.139} C_VEL
LIN {X 0,Y 545.082,Z 311.587,A -85,B 0,C 180,E1 -3733.105,E2 -3733.105} C_VEL
LIN {X 0,Y 545.044,Z 311.59,A -85,B 0,C 180,E1 -3736.225,E2 -3736.225} C_VEL
LIN {X 0,Y 545.021,Z 311.599,A -85,B 0,C 180,E1 -3738.88,E2 -3738.88} C_VEL
LIN {X 0,Y 545.073,Z 311.59,A -85,B 0,C 180,E1 -3740.818,E2 -3740.818} C_VEL
LIN {X 0,Y 545.049,Z 311.591,A -85,B 0,C 180,E1 -3743.62,E2 -3743.62} C_VEL
LIN {X 0,Y 545.063,Z 311.588,A -85,B 0,C 180,E1 -3746.328,E2 -3746.328} C_VEL
LIN {X 0,Y 545.055,Z 311.593,A -85,B 0,C 180,E1 -3748.951,E2 -3748.951} C_VEL
LIN {X 0,Y 545.029,Z 311.592,A -85,B 0,C 180,E1 -3751.503,E2 -3751.503} C_VEL
LIN {X 0,Y 545.064,Z 311.589,A -85,B 0,C 180,E1 -3753.999,E2 -3753.999} C_VEL
LIN {X 0,Y 545.082,Z 311.587,A -85,B 0,C 180,E1 -3756.441,E2 -3756.441} C_VEL
LIN {X 0,Y 545.09,Z 311.589,A -85,B 0,C 180,E1 -3759.628,E2 -3759.628} C_VEL
LIN {X 0,Y 545.079,Z 311.591,A -85,B 0,C 180,E1 -3762.749,E2 -3762.749} C_VEL
LIN {X 0,Y 545.069,Z 311.588,A -85,B 0,C 180,E1 -3765.819,E2 -3765.819} C_VEL
LIN {X 0,Y 545.107,Z 311.581,A -85,B 0,C 180,E1 -3768.849,E2 -3768.849} C_VEL
LIN {X 0,Y 545.125,Z 311.582,A -85,B 0,C 180,E1 -3771.847,E2 -3771.847} C_VEL
LIN {X 0,Y 545.2,Z 311.575,A -85,B 0,C 180,E1 -3774.823,E2 -3774.823} C_VEL
LIN {X 0,Y 545.188,Z 311.573,A -85,B 0,C 180,E1 -3777.784,E2 -3777.784} C_VEL
LIN {X 0,Y 545.189,Z 311.571,A -85,B 0,C 180,E1 -3780.739,E2 -3780.739} C_VEL
LIN {X 0,Y 545.157,Z 311.576,A -85,B 0,C 180,E1 -3782.956,E2 -3782.956} C_VEL
LIN {X 0,Y 545.176,Z 311.573,A -85,B 0,C 180,E1 -3785.92,E2 -3785.92} C_VEL
LIN {X 0,Y 545.118,Z 311.584,A -85,B 0,C 180,E1 -3788.9,E2 -3788.9} C_VEL
LIN {X 0,Y 545.092,Z 311.59,A -85,B 0,C 180,E1 -3791.905,E2 -3791.905} C_VEL
LIN {X 0,Y 545.069,Z 311.588,A -85,B 0,C 180,E1 -3794.944,E2 -3794.944} C_VEL
LIN {X 0,Y 545.072,Z 311.586,A -85,B 0,C 180,E1 -3798.026,E2 -3798.026} C_VEL
LIN {X 0,Y 545.09,Z 311.588,A -85,B 0,C 180,E1 -3800.372,E2 -3800.372} C_VEL
LIN {X 0,Y 545.082,Z 311.587,A -85,B 0,C 180,E1 -3803.559,E2 -3803.559} C_VEL
LIN {X 0,Y 545.064,Z 311.591,A -85,B 0,C 180,E1 -3806.001,E2 -3806.001} C_VEL
LIN {X 0,Y 545.035,Z 311.593,A -85,B 0,C 180,E1 -3808.74,E2 -3808.74} C_VEL
LIN {X 0,Y 545.051,Z 311.588,A -85,B 0,C 180,E1 -3811.68,E2 -3811.68} C_VEL
LIN {X 0,Y 545.074,Z 311.59,A -85,B 0,C 180,E1 -3814.564,E2 -3814.564} C_VEL
LIN {X 0,Y 545.058,Z 311.589,A -85,B 0,C 180,E1 -3817.015,E2 -3817.015} C_VEL
LIN {X 0,Y 544.351,Z 311.681,A -85,B 0,C 180,E1 -3817.632,E2 -3817.632} C_VEL
LIN {X 0,Y 541.49,Z 312.035,A -85,B 0,C 180,E1 -3818.633,E2 -3818.633} C_VEL
LIN {X 0,Y 539.097,Z 312.335,A -85,B 0,C 180,E1 -3819.438,E2 -3819.438} C_VEL
LIN {X 0,Y 538.072,Z 312.459,A -85,B 0,C 180,E1 -3820.06,E2 -3820.06} C_VEL
LIN {X 0,Y 537.989,Z 312.469,A -85,B 0,C 180,E1 -3820.271,E2 -3820.271} C_VEL
LIN {X 0,Y 537.972,Z 312.474,A -85,B 0,C 180,E1 -3822.983,E2 -3822.983} C_VEL
LIN {X 0,Y 538.019,Z 312.466,A -85,B 0,C 180,E1 -3825.927,E2 -3825.927} C_VEL
LIN {X 0,Y 538.075,Z 312.46,A -85,B 0,C 180,E1 -3829.25,E2 -3829.25} C_VEL
LIN {X 0,Y 537.988,Z 312.469,A -85,B 0,C 180,E1 -3832.123,E2 -3832.123} C_VEL
LIN {X 0,Y 537.946,Z 312.475,A -85,B 0,C 180,E1 -3834.096,E2 -3834.096} C_VEL
LIN {X 0,Y 537.925,Z 312.821,A -85,B 0,C 180,E1 -3834.911,E2 -3834.911} C_VEL
LIN {X 0,Y 537.928,Z 316.985,A -85,B 0,C 180,E1 -3837.612,E2 -3837.612} C_VEL
LIN {X 0,Y 537.843,Z 321.079,A -85,B 0,C 180,E1 -3840.229,E2 -3840.229} C_VEL
LIN {X 0,Y 537.788,Z 325.145,A -85,B 0,C 180,E1 -3842.782,E2 -3842.782} C_VEL
LIN {X 0,Y 537.771,Z 329.212,A -85,B 0,C 180,E1 -3845.28,E2 -3845.28} C_VEL
LIN {X 0,Y 537.687,Z 334.623,A -85,B 0,C 180,E1 -3848.533,E2 -3848.533} C_VEL
LIN {X 0,Y 537.645,Z 338.706,A -85,B 0,C 180,E1 -3850.926,E2 -3850.926} C_VEL
LIN {X 0,Y 537.587,Z 342.707,A -85,B 0,C 180,E1 -3853.286,E2 -3853.286} C_VEL
LIN {X 0,Y 537.604,Z 346.726,A -85,B 0,C 180,E1 -3855.619,E2 -3855.619} C_VEL
LIN {X 0,Y 537.546,Z 348.661,A -85,B 0,C 180,E1 -3856.726,E2 -3856.726} C_VEL
LIN {X 0,Y 539.197,Z 359.315,A -85,B 0,C 180,E1 -3857.031,E2 -3857.031} C_VEL
LIN {X 0,Y 538.959,Z 372.261,A -85,B 0,C 180,E1 -3857.48,E2 -3857.48} C_VEL
LIN {X 0,Y 538.716,Z 384.782,A -85,B 0,C 180,E1 -3858.081,E2 -3858.081} C_VEL
LIN {X 0,Y 538.529,Z 396.317,A -85,B 0,C 180,E1 -3858.807,E2 -3858.807} C_VEL
LIN {X 0,Y 538.316,Z 407.034,A -85,B 0,C 180,E1 -3859.659,E2 -3859.659} C_VEL
LIN {X 0,Y 538.086,Z 416.696,A -85,B 0,C 180,E1 -3860.604,E2 -3860.604} C_VEL
LIN {X 0,Y 537.922,Z 424.613,A -85,B 0,C 180,E1 -3861.548,E2 -3861.548} C_VEL
LIN {X 0,Y 537.759,Z 432.359,A -85,B 0,C 180,E1 -3862.68,E2 -3862.68} C_VEL
LIN {X 0,Y 537.694,Z 439.464,A -85,B 0,C 180,E1 -3863.998,E2 -3863.998} C_VEL
LIN {X 0,Y 537.54,Z 444.203,A -85,B 0,C 180,E1 -3865.125,E2 -3865.125} C_VEL
LIN {X 0,Y 537.591,Z 447.834,A -85,B 0,C 180,E1 -3866.253,E2 -3866.253} C_VEL
LIN {X 0,Y 537.551,Z 449.71,A -85,B 0,C 180,E1 -3867.003,E2 -3867.003} C_VEL
LIN {X 0,Y 537.49,Z 451.129,A -85,B 0,C 180,E1 -3867.752,E2 -3867.752} C_VEL
LIN {X 0,Y 537.442,Z 452.757,A -85,B 0,C 180,E1 -3869.251,E2 -3869.251} C_VEL
LIN {X 0,Y 537.442,Z 452.996,A -85,B 0,C 180,E1 -3870,E2 -3870} C_VEL
LIN {X 0,Y 537.442,Z 452.814,A -85,B 0,C 180,E1 -3870.75,E2 -3870.75} C_VEL
LIN {X 0,Y 537.491,Z 451.26,A -85,B 0,C 180,E1 -3872.248,E2 -3872.248} C_VEL
LIN {X 0,Y 537.552,Z 449.899,A -85,B 0,C 180,E1 -3872.998,E2 -3872.998} C_VEL
LIN {X 0,Y 537.604,Z 447.021,A -85,B 0,C 180,E1 -3874.123,E2 -3874.123} C_VEL
LIN {X 0,Y 537.587,Z 443.119,A -85,B 0,C 180,E1 -3875.251,E2 -3875.251} C_VEL
LIN {X 0,Y 537.639,Z 438.365,A -85,B 0,C 180,E1 -3876.321,E2 -3876.321} C_VEL
LIN {X 0,Y 537.79,Z 431.755,A -85,B 0,C 180,E1 -3877.509,E2 -3877.509} C_VEL
LIN {X 0,Y 537.952,Z 423.829,A -85,B 0,C 180,E1 -3878.641,E2 -3878.641} C_VEL
LIN {X 0,Y 538.133,Z 413.972,A -85,B 0,C 180,E1 -3879.775,E2 -3879.775} C_VEL
LIN {X 0,Y 538.385,Z 403.644,A -85,B 0,C 180,E1 -3880.721,E2 -3880.721} C_VEL
LIN {X 0,Y 538.578,Z 392.887,A -85,B 0,C 180,E1 -3881.516,E2 -3881.516} C_VEL
LIN {X 0,Y 538.761,Z 382.293,A -85,B 0,C 180,E1 -3882.143,E2 -3882.143} C_VEL
LIN {X 0,Y 539.04,Z 369.777,A -85,B 0,C 180,E1 -3882.71,E2 -3882.71} C_VEL
LIN {X 0,Y 539.066,Z 357.257,A -85,B 0,C 180,E1 -3883.117,E2 -3883.117} C_VEL
LIN {X 0,Y 537.556,Z 348.663,A -85,B 0,C 180,E1 -3883.371,E2 -3883.371} C_VEL
LIN {X 0,Y 537.572,Z 344.227,A -85,B 0,C 180,E1 -3885.935,E2 -3885.935} C_VEL
LIN {X 0,Y 537.624,Z 338.866,A -85,B 0,C 180,E1 -3889.075,E2 -3889.075} C_VEL
LIN {X 0,Y 537.687,Z 333.42,A -85,B 0,C 180,E1 -3892.275,E2 -3892.275} C_VEL
LIN {X 0,Y 537.769,Z 329.359,A -85,B 0,C 180,E1 -3894.721,E2 -3894.721} C_VEL
LIN {X 0,Y 537.82,Z 323.935,A -85,B 0,C 180,E1 -3898.062,E2 -3898.062} C_VEL
LIN {X 0,Y 537.85,Z 319.865,A -85,B 0,C 180,E1 -3900.637,E2 -3900.637} C_VEL
LIN {X 0,Y 537.981,Z 315.752,A -85,B 0,C 180,E1 -3903.276,E2 -3903.276} C_VEL
LIN {X 0,Y 537.964,Z 312.96,A -85,B 0,C 180,E1 -3905.087,E2 -3905.087} C_VEL
LIN {X 0,Y 537.955,Z 312.473,A -85,B 0,C 180,E1 -3906.007,E2 -3906.007} C_VEL
LIN {X 0,Y 538.01,Z 312.471,A -85,B 0,C 180,E1 -3908.83,E2 -3908.83} C_VEL
LIN {X 0,Y 538.037,Z 312.466,A -85,B 0,C 180,E1 -3911.772,E2 -3911.772} C_VEL
LIN {X 0,Y 538.005,Z 312.466,A -85,B 0,C 180,E1 -3914.862,E2 -3914.862} C_VEL
LIN {X 0,Y 537.971,Z 312.476,A -85,B 0,C 180,E1 -3917.209,E2 -3917.209} C_VEL
LIN {X 0,Y 538.005,Z 312.469,A -85,B 0,C 180,E1 -3920.201,E2 -3920.201} C_VEL
LIN {X 0,Y 538.026,Z 312.465,A -85,B 0,C 180,E1 -3923.067,E2 -3923.067} C_VEL
LIN {X 0,Y 538.022,Z 312.469,A -85,B 0,C 180,E1 -3925.827,E2 -3925.827} C_VEL
LIN {X 0,Y 538.006,Z 312.466,A -85,B 0,C 180,E1 -3928.498,E2 -3928.498} C_VEL
LIN {X 0,Y 537.996,Z 312.472,A -85,B 0,C 180,E1 -3931.096,E2 -3931.096} C_VEL
LIN {X 0,Y 538.007,Z 312.467,A -85,B 0,C 180,E1 -3933.631,E2 -3933.631} C_VEL
LIN {X 0,Y 538.002,Z 312.472,A -85,B 0,C 180,E1 -3936.122,E2 -3936.122} C_VEL
LIN {X 0,Y 538.038,Z 312.468,A -85,B 0,C 180,E1 -3939.348,E2 -3939.348} C_VEL
LIN {X 0,Y 538.05,Z 312.463,A -85,B 0,C 180,E1 -3942.517,E2 -3942.517} C_VEL
LIN {X 0,Y 538.046,Z 312.461,A -85,B 0,C 180,E1 -3945.63,E2 -3945.63} C_VEL
LIN {X 0,Y 538.071,Z 312.459,A -85,B 0,C 180,E1 -3948.701,E2 -3948.701} C_VEL
LIN {X 0,Y 538.082,Z 312.461,A -85,B 0,C 180,E1 -3951.739,E2 -3951.739} C_VEL
LIN {X 0,Y 538.161,Z 312.452,A -85,B 0,C 180,E1 -3954.755,E2 -3954.755} C_VEL
LIN {X 0,Y 538.163,Z 312.447,A -85,B 0,C 180,E1 -3957.755,E2 -3957.755} C_VEL
LIN {X 0,Y 538.164,Z 312.447,A -85,B 0,C 180,E1 -3960.748,E2 -3960.748} C_VEL
LIN {X 0,Y 538.127,Z 312.453,A -85,B 0,C 180,E1 -3962.994,E2 -3962.994} C_VEL
LIN {X 0,Y 538.13,Z 312.452,A -85,B 0,C 180,E1 -3965.997,E2 -3965.997} C_VEL
LIN {X 0,Y 538.071,Z 312.46,A -85,B 0,C 180,E1 -3969.018,E2 -3969.018} C_VEL
LIN {X 0,Y 538.055,Z 312.466,A -85,B 0,C 180,E1 -3972.063,E2 -3972.063} C_VEL
LIN {X 0,Y 538.034,Z 312.466,A -85,B 0,C 180,E1 -3975.144,E2 -3975.144} C_VEL
LIN {X 0,Y 538.025,Z 312.465,A -85,B 0,C 180,E1 -3978.27,E2 -3978.27} C_VEL
LIN {X 0,Y 538.038,Z 312.467,A -85,B 0,C 180,E1 -3980.651,E2 -3980.651} C_VEL
LIN {X 0,Y 538.02,Z 312.47,A -85,B 0,C 180,E1 -3983.888,E2 -3983.888} C_VEL
LIN {X 0,Y 538.012,Z 312.465,A -85,B 0,C 180,E1 -3986.368,E2 -3986.368} C_VEL
LIN {X 0,Y 537.987,Z 312.472,A -85,B 0,C 180,E1 -3988.926,E2 -3988.926} C_VEL
LIN {X 0,Y 538.011,Z 312.467,A -85,B 0,C 180,E1 -3991.888,E2 -3991.888} C_VEL
LIN {X 0,Y 538.024,Z 312.468,A -85,B 0,C 180,E1 -3994.62,E2 -3994.62} C_VEL
LIN {X 0,Y 538.004,Z 312.468,A -85,B 0,C 180,E1 -3997.171,E2 -3997.171} C_VEL
LIN {X 0,Y 538.017,Z 312.466,A -85,B 0,C 180,E1 -3999.798,E2 -3999.798} C_VEL
LIN {X 0,Y 537.968,Z 312.477,A -85,B 0,C 180,E1 -4002.982,E2 -4002.982} C_VEL
LIN {X 0,Y 538.017,Z 312.468,A -85,B 0,C 180,E1 -4005.927,E2 -4005.927} C_VEL
LIN {X 0,Y 538.036,Z 312.467,A -85,B 0,C 180,E1 -4008.228,E2 -4008.228} C_VEL
LIN {X 0,Y 538.011,Z 312.472,A -85,B 0,C 180,E1 -4011.17,E2 -4011.17} C_VEL
LIN {X 0,Y 538.062,Z 312.633,A -85,B 0,C 180,E1 -4012.822,E2 -4012.822} C_VEL
LIN {X 0,Y 538.598,Z 317.743,A -85,B 0,C 180,E1 -4014.961,E2 -4014.961} C_VEL
LIN {X 0,Y 538.472,Z 324.489,A -85,B 0,C 180,E1 -4017.648,E2 -4017.648} C_VEL
LIN {X 0,Y 538.357,Z 331.205,A -85,B 0,C 180,E1 -4020.26,E2 -4020.26} C_VEL
LIN {X 0,Y 538.18,Z 338.996,A -85,B 0,C 180,E1 -4023.223,E2 -4023.223} C_VEL
LIN {X 0,Y 538.081,Z 346.787,A -85,B 0,C 180,E1 -4026.115,E2 -4026.115} C_VEL
LIN {X 0,Y 537.947,Z 354.579,A -85,B 0,C 180,E1 -4028.945,E2 -4028.945} C_VEL
LIN {X 0,Y 537.831,Z 362.37,A -85,B 0,C 180,E1 -4031.723,E2 -4031.723} C_VEL
LIN {X 0,Y 537.763,Z 371.274,A -85,B 0,C 180,E1 -4034.848,E2 -4034.848} C_VEL
LIN {X 0,Y 537.699,Z 376.491,A -85,B 0,C 180,E1 -4036.657,E2 -4036.657} C_VEL
LIN {X 0,Y 539.248,Z 386.35,A -85,B 0,C 180,E1 -4036.912,E2 -4036.912} C_VEL
LIN {X 0,Y 539.085,Z 398.472,A -85,B 0,C 180,E1 -4037.291,E2 -4037.291} C_VEL
LIN {X 0,Y 538.838,Z 409.485,A -85,B 0,C 180,E1 -4037.763,E2 -4037.763} C_VEL
LIN {X 0,Y 538.65,Z 420.427,A -85,B 0,C 180,E1 -4038.372,E2 -4038.372} C_VEL
LIN {X 0,Y 538.414,Z 431.924,A -85,B 0,C 180,E1 -4039.185,E2 -4039.185} C_VEL
LIN {X 0,Y 538.2,Z 441.6,A -85,B 0,C 180,E1 -4040.036,E2 -4040.036} C_VEL
LIN {X 0,Y 538.015,Z 450.412,A -85,B 0,C 180,E1 -4040.981,E2 -4040.981} C_VEL
LIN {X 0,Y 537.829,Z 459,A -85,B 0,C 180,E1 -4042.114,E2 -4042.114} C_VEL
LIN {X 0,Y 537.705,Z 465.867,A -85,B 0,C 180,E1 -4043.244,E2 -4043.244} C_VEL
LIN {X 0,Y 537.676,Z 471.365,A -85,B 0,C 180,E1 -4044.374,E2 -4044.374} C_VEL
LIN {X 0,Y 537.558,Z 475.677,A -85,B 0,C 180,E1 -4045.501,E2 -4045.501} C_VEL
LIN {X 0,Y 537.591,Z 477.957,A -85,B 0,C 180,E1 -4046.252,E2 -4046.252} C_VEL
LIN {X 0,Y 537.551,Z 479.808,A -85,B 0,C 180,E1 -4047.002,E2 -4047.002} C_VEL
LIN {X 0,Y 537.49,Z 481.198,A -85,B 0,C 180,E1 -4047.752,E2 -4047.752} C_VEL
LIN {X 0,Y 537.442,Z 482.785,A -85,B 0,C 180,E1 -4049.25,E2 -4049.25} C_VEL
LIN {X 0,Y 537.442,Z 483,A -85,B 0,C 180,E1 -4050,E2 -4050} C_VEL
LIN {X 0,Y 537.451,Z 482.187,A -85,B 0,C 180,E1 -4051.498,E2 -4051.498} C_VEL
LIN {X 0,Y 537.49,Z 481.2,A -85,B 0,C 180,E1 -4052.248,E2 -4052.248} C_VEL
LIN {X 0,Y 537.551,Z 479.811,A -85,B 0,C 180,E1 -4052.997,E2 -4052.997} C_VEL
LIN {X 0,Y 537.603,Z 476.897,A -85,B 0,C 180,E1 -4054.123,E2 -4054.123} C_VEL
LIN {X 0,Y 537.587,Z 472.951,A -85,B 0,C 180,E1 -4055.25,E2 -4055.25} C_VEL
LIN {X 0,Y 537.649,Z 468.1,A -85,B 0,C 180,E1 -4056.331,E2 -4056.331} C_VEL
LIN {X 0,Y 537.79,Z 461.472,A -85,B 0,C 180,E1 -4057.509,E2 -4057.509} C_VEL
LIN {X 0,Y 537.972,Z 453.482,A -85,B 0,C 180,E1 -4058.64,E2 -4058.64} C_VEL
LIN {X 0,Y 538.118,Z 445.341,A -85,B 0,C 180,E1 -4059.585,E2 -4059.585} C_VEL
LIN {X 0,Y 538.374,Z 435.407,A -85,B 0,C 180,E1 -4060.53,E2 -4060.53} C_VEL
LIN {X 0,Y 538.541,Z 425.595,A -85,B 0,C 180,E1 -4061.288,E2 -4061.288} C_VEL
LIN {X 0,Y 538.739,Z 414.605,A -85,B 0,C 180,E1 -4061.97,E2 -4061.97} C_VEL
LIN {X 0,Y 538.944,Z 402.124,A -85,B 0,C 180,E1 -4062.568,E2 -4062.568} C_VEL
LIN {X 0,Y 539.199,Z 389.112,A -85,B 0,C 180,E1 -4063.017,E2 -4063.017} C_VEL
LIN {X 0,Y 538.945,Z 384.063,A -85,B 0,C 180,E1 -4063.155,E2 -4063.155} C_VEL
LIN {X 0,Y 537.698,Z 376.493,A -85,B 0,C 180,E1 -4063.342,E2 -4063.342} C_VEL
LIN {X 0,Y 537.762,Z 369.05,A -85,B 0,C 180,E1 -4065.928,E2 -4065.928} C_VEL
LIN {X 0,Y 537.847,Z 361.259,A -85,B 0,C 180,E1 -4068.671,E2 -4068.671} C_VEL
LIN {X 0,Y 537.984,Z 353.467,A -85,B 0,C 180,E1 -4071.455,E2 -4071.455} C_VEL
LIN {X 0,Y 538.097,Z 345.677,A -85,B 0,C 180,E1 -4074.293,E2 -4074.293} C_VEL
LIN {X 0,Y 538.257,Z 337.356,A -85,B 0,C 180,E1 -4077.392,E2 -4077.392} C_VEL
LIN {X 0,Y 538.377,Z 329.229,A -85,B 0,C 180,E1 -4080.507,E2 -4080.507} C_VEL
LIN {X 0,Y 538.526,Z 321.93,A -85,B 0,C 180,E1 -4083.36,E2 -4083.36} C_VEL
LIN {X 0,Y 538.599,Z 316.608,A -85,B 0,C 180,E1 -4085.496,E2 -4085.496} C_VEL
LIN {X 0,Y 538.044,Z 312.468,A -85,B 0,C 180,E1 -4087.3,E2 -4087.3} C_VEL
LIN {X 0,Y 538.05,Z 312.464,A -85,B 0,C 180,E1 -4089.793,E2 -4089.793} C_VEL
LIN {X 0,Y 538.019,Z 312.467,A -85,B 0,C 180,E1 -4092.785,E2 -4092.785} C_VEL
LIN {X 0,Y 538.026,Z 312.467,A -85,B 0,C 180,E1 -4095.14,E2 -4095.14} C_VEL
LIN {X 0,Y 537.991,Z 312.468,A -85,B 0,C 180,E1 -4098.223,E2 -4098.223} C_VEL
LIN {X 0,Y 538.005,Z 312.467,A -85,B 0,C 180,E1 -4101.169,E2 -4101.169} C_VEL
LIN {X 0,Y 538.022,Z 312.47,A -85,B 0,C 180,E1 -4104.083,E2 -4104.083} C_VEL
LIN {X 0,Y 538.024,Z 312.465,A -85,B 0,C 180,E1 -4106.727,E2 -4106.727} C_VEL
LIN {X 0,Y 537.999,Z 312.47,A -85,B 0,C 180,E1 -4109.559,E2 -4109.559} C_VEL
LIN {X 0,Y 538.015,Z 312.468,A -85,B 0,C 180,E1 -4112.793,E2 -4112.793} C_VEL
LIN {X 0,Y 538.015,Z 312.465,A -85,B 0,C 180,E1 -4115.291,E2 -4115.291} C_VEL
LIN {X 0,Y 538.006,Z 312.47,A -85,B 0,C 180,E1 -4118.041,E2 -4118.041} C_VEL
LIN {X 0,Y 538.031,Z 312.468,A -85,B 0,C 180,E1 -4120.94,E2 -4120.94} C_VEL
LIN {X 0,Y 538.003,Z 312.469,A -85,B 0,C 180,E1 -4123.298,E2 -4123.298} C_VEL
LIN {X 0,Y 538.038,Z 312.463,A -85,B 0,C 180,E1 -4125.63,E2 -4125.63} C_VEL
LIN {X 0,Y 538.066,Z 312.458,A -85,B 0,C 180,E1 -4128.701,E2 -4128.701} C_VEL
LIN {X 0,Y 538.081,Z 312.46,A -85,B 0,C 180,E1 -4131.74,E2 -4131.74} C_VEL
LIN {X 0,Y 538.177,Z 312.45,A -85,B 0,C 180,E1 -4134.755,E2 -4134.755} C_VEL
LIN {X 0,Y 538.159,Z 312.449,A -85,B 0,C 180,E1 -4137.755,E2 -4137.755} C_VEL
LIN {X 0,Y 538.16,Z 312.447,A -85,B 0,C 180,E1 -4140.748,E2 -4140.748} C_VEL
LIN {X 0,Y 538.125,Z 312.452,A -85,B 0,C 180,E1 -4142.995,E2 -4142.995} C_VEL
LIN {X 0,Y 538.126,Z 312.452,A -85,B 0,C 180,E1 -4145.997,E2 -4145.997} C_VEL
LIN {X 0,Y 538.067,Z 312.461,A -85,B 0,C 180,E1 -4149.018,E2 -4149.018} C_VEL
LIN {X 0,Y 538.051,Z 312.465,A -85,B 0,C 180,E1 -4152.063,E2 -4152.063} C_VEL
LIN {X 0,Y 538.03,Z 312.466,A -85,B 0,C 180,E1 -4155.144,E2 -4155.144} C_VEL
LIN {X 0,Y 538.024,Z 312.464,A -85,B 0,C 180,E1 -4158.271,E2 -4158.271} C_VEL
LIN {X 0,Y 538.034,Z 312.469,A -85,B 0,C 180,E1 -4160.652,E2 -4160.652} C_VEL
LIN {X 0,Y 538.015,Z 312.47,A -85,B 0,C 180,E1 -4163.888,E2 -4163.888} C_VEL
LIN {X 0,Y 538.025,Z 312.465,A -85,B 0,C 180,E1 -4166.368,E2 -4166.368} C_VEL
LIN {X 0,Y 537.982,Z 312.474,A -85,B 0,C 180,E1 -4168.926,E2 -4168.926} C_VEL
LIN {X 0,Y 538.006,Z 312.466,A -85,B 0,C 180,E1 -4171.889,E2 -4171.889} C_VEL
LIN {X 0,Y 538.024,Z 312.467,A -85,B 0,C 180,E1 -4174.622,E2 -4174.622} C_VEL
LIN {X 0,Y 538.001,Z 312.469,A -85,B 0,C 180,E1 -4177.171,E2 -4177.171} C_VEL
LIN {X 0,Y 538.016,Z 312.468,A -85,B 0,C 180,E1 -4179.798,E2 -4179.798} C_VEL
LIN {X 0,Y 537.989,Z 312.469,A -85,B 0,C 180,E1 -4180.271,E2 -4180.271} C_VEL
LIN {X 0,Y 537.321,Z 312.556,A -85,B 0,C 180,E1 -4180.896,E2 -4180.896} C_VEL
LIN {X 0,Y 534.465,Z 312.909,A -85,B 0,C 180,E1 -4181.911,E2 -4181.911} C_VEL
LIN {X 0,Y 532.051,Z 313.214,A -85,B 0,C 180,E1 -4182.728,E2 -4182.728} C_VEL
LIN {X 0,Y 531.015,Z 313.338,A -85,B 0,C 180,E1 -4183.359,E2 -4183.359} C_VEL
LIN {X 0,Y 530.93,Z 313.347,A -85,B 0,C 180,E1 -4183.572,E2 -4183.572} C_VEL
LIN {X 0,Y 530.955,Z 313.349,A -85,B 0,C 180,E1 -4186.506,E2 -4186.506} C_VEL
LIN {X 0,Y 531.023,Z 313.34,A -85,B 0,C 180,E1 -4189.572,E2 -4189.572} C_VEL
LIN {X 0,Y 530.963,Z 313.345,A -85,B 0,C 180,E1 -4192.578,E2 -4192.578} C_VEL
LIN {X 0,Y 530.879,Z 313.357,A -85,B 0,C 180,E1 -4194.375,E2 -4194.375} C_VEL
LIN {X 0,Y 530.941,Z 314.292,A -85,B 0,C 180,E1 -4195.308,E2 -4195.308} C_VEL
LIN {X 0,Y 530.888,Z 318.443,A -85,B 0,C 180,E1 -4198.028,E2 -4198.028} C_VEL
LIN {X 0,Y 530.794,Z 322.926,A -85,B 0,C 180,E1 -4200.913,E2 -4200.913} C_VEL
LIN {X 0,Y 530.689,Z 326.613,A -85,B 0,C 180,E1 -4203.24,E2 -4203.24} C_VEL
LIN {X 0,Y 530.7,Z 331.121,A -85,B 0,C 180,E1 -4206.031,E2 -4206.031} C_VEL
LIN {X 0,Y 530.579,Z 336.109,A -85,B 0,C 180,E1 -4209.045,E2 -4209.045} C_VEL
LIN {X 0,Y 530.525,Z 340.199,A -85,B 0,C 180,E1 -4211.463,E2 -4211.463} C_VEL
LIN {X 0,Y 530.488,Z 344.205,A -85,B 0,C 180,E1 -4213.847,E2 -4213.847} C_VEL
LIN {X 0,Y 530.485,Z 348.577,A -85,B 0,C 180,E1 -4216.4,E2 -4216.4} C_VEL
LIN {X 0,Y 530.48,Z 348.833,A -85,B 0,C 180,E1 -4216.546,E2 -4216.546} C_VEL
LIN {X 0,Y 532.282,Z 359.552,A -85,B 0,C 180,E1 -4216.86,E2 -4216.86} C_VEL
LIN {X 0,Y 532.047,Z 372.49,A -85,B 0,C 180,E1 -4217.315,E2 -4217.315} C_VEL
LIN {X 0,Y 531.806,Z 384.293,A -85,B 0,C 180,E1 -4217.885,E2 -4217.885} C_VEL
LIN {X 0,Y 531.614,Z 395.178,A -85,B 0,C 180,E1 -4218.563,E2 -4218.563} C_VEL
LIN {X 0,Y 531.352,Z 406.17,A -85,B 0,C 180,E1 -4219.426,E2 -4219.426} C_VEL
LIN {X 0,Y 531.072,Z 416.857,A -85,B 0,C 180,E1 -4220.479,E2 -4220.479} C_VEL
LIN {X 0,Y 530.891,Z 424.736,A -85,B 0,C 180,E1 -4221.436,E2 -4221.436} C_VEL
LIN {X 0,Y 530.722,Z 432.442,A -85,B 0,C 180,E1 -4222.582,E2 -4222.582} C_VEL
LIN {X 0,Y 530.606,Z 439.507,A -85,B 0,C 180,E1 -4223.918,E2 -4223.918} C_VEL
LIN {X 0,Y 530.459,Z 444.218,A -85,B 0,C 180,E1 -4225.06,E2 -4225.06} C_VEL
LIN {X 0,Y 530.516,Z 447.835,A -85,B 0,C 180,E1 -4226.203,E2 -4226.203} C_VEL
LIN {X 0,Y 530.457,Z 449.712,A -85,B 0,C 180,E1 -4226.963,E2 -4226.963} C_VEL
LIN {X 0,Y 530.412,Z 451.129,A -85,B 0,C 180,E1 -4227.722,E2 -4227.722} C_VEL
LIN {X 0,Y 530.344,Z 452.757,A -85,B 0,C 180,E1 -4229.241,E2 -4229.241} C_VEL
LIN {X 0,Y 530.343,Z 452.997,A -85,B 0,C 180,E1 -4230,E2 -4230} C_VEL
LIN {X 0,Y 530.344,Z 452.813,A -85,B 0,C 180,E1 -4230.76,E2 -4230.76} C_VEL
LIN {X 0,Y 530.412,Z 451.259,A -85,B 0,C 180,E1 -4232.278,E2 -4232.278} C_VEL
LIN {X 0,Y 530.457,Z 449.897,A -85,B 0,C 180,E1 -4233.038,E2 -4233.038} C_VEL
LIN {X 0,Y 530.523,Z 447.019,A -85,B 0,C 180,E1 -4234.179,E2 -4234.179} C_VEL
LIN {X 0,Y 530.524,Z 443.135,A -85,B 0,C 180,E1 -4235.321,E2 -4235.321} C_VEL
LIN {X 0,Y 530.593,Z 437.583,A -85,B 0,C 180,E1 -4236.576,E2 -4236.576} C_VEL
LIN {X 0,Y 530.758,Z 430.612,A -85,B 0,C 180,E1 -4237.801,E2 -4237.801} C_VEL
LIN {X 0,Y 530.903,Z 422.47,A -85,B 0,C 180,E1 -4238.949,E2 -4238.949} C_VEL
LIN {X 0,Y 531.124,Z 414.134,A -85,B 0,C 180,E1 -4239.905,E2 -4239.905} C_VEL
LIN {X 0,Y 531.403,Z 403.843,A -85,B 0,C 180,E1 -4240.863,E2 -4240.863} C_VEL
LIN {X 0,Y 531.63,Z 392.398,A -85,B 0,C 180,E1 -4241.716,E2 -4241.716} C_VEL
LIN {X 0,Y 531.883,Z 380.686,A -85,B 0,C 180,E1 -4242.399,E2 -4242.399} C_VEL
LIN {X 0,Y 532.161,Z 368.677,A -85,B 0,C 180,E1 -4242.926,E2 -4242.926} C_VEL
LIN {X 0,Y 532.127,Z 358.137,A -85,B 0,C 180,E1 -4243.272,E2 -4243.272} C_VEL
LIN {X 0,Y 530.471,Z 348.837,A -85,B 0,C 180,E1 -4243.552,E2 -4243.552} C_VEL
LIN {X 0,Y 530.502,Z 345.739,A -85,B 0,C 180,E1 -4245.364,E2 -4245.364} C_VEL
LIN {X 0,Y 530.516,Z 340.358,A -85,B 0,C 180,E1 -4248.538,E2 -4248.538} C_VEL
LIN {X 0,Y 530.58,Z 336.258,A -85,B 0,C 180,E1 -4250.955,E2 -4250.955} C_VEL
LIN {X 0,Y 530.686,Z 331.275,A -85,B 0,C 180,E1 -4253.966,E2 -4253.966} C_VEL
LIN {X 0,Y 530.69,Z 326.756,A -85,B 0,C 180,E1 -4256.761,E2 -4256.761} C_VEL
LIN {X 0,Y 530.79,Z 322.685,A -85,B 0,C 180,E1 -4259.334,E2 -4259.334} C_VEL
LIN {X 0,Y 530.881,Z 318.413,A -85,B 0,C 180,E1 -4262.085,E2 -4262.085} C_VEL
LIN {X 0,Y 530.941,Z 314.2,A -85,B 0,C 180,E1 -4264.846,E2 -4264.846} C_VEL
LIN {X 0,Y 530.895,Z 313.355,A -85,B 0,C 180,E1 -4265.624,E2 -4265.624} C_VEL
LIN {X 0,Y 530.954,Z 313.35,A -85,B 0,C 180,E1 -4268.471,E2 -4268.471} C_VEL
LIN {X 0,Y 530.997,Z 313.34,A -85,B 0,C 180,E1 -4271.435,E2 -4271.435} C_VEL
LIN {X 0,Y 530.974,Z 313.341,A -85,B 0,C 180,E1 -4274.548,E2 -4274.548} C_VEL
LIN {X 0,Y 530.916,Z 313.353,A -85,B 0,C 180,E1 -4277.537,E2 -4277.537} C_VEL
LIN {X 0,Y 530.966,Z 313.347,A -85,B 0,C 180,E1 -4280.555,E2 -4280.555} C_VEL
LIN {X 0,Y 530.965,Z 313.345,A -85,B 0,C 180,E1 -4283.442,E2 -4283.442} C_VEL
LIN {X 0,Y 530.997,Z 313.34,A -85,B 0,C 180,E1 -4286.494,E2 -4286.494} C_VEL
LIN {X 0,Y 530.959,Z 313.349,A -85,B 0,C 180,E1 -4289.357,E2 -4289.357} C_VEL
LIN {X 0,Y 530.957,Z 313.348,A -85,B 0,C 180,E1 -4292.478,E2 -4292.478} C_VEL
LIN {X 0,Y 530.956,Z 313.346,A -85,B 0,C 180,E1 -4294.94,E2 -4294.94} C_VEL
LIN {X 0,Y 530.973,Z 313.347,A -85,B 0,C 180,E1 -4297.898,E2 -4297.898} C_VEL
LIN {X 0,Y 530.99,Z 313.342,A -85,B 0,C 180,E1 -4300.677,E2 -4300.677} C_VEL
LIN {X 0,Y 530.977,Z 313.346,A -85,B 0,C 180,E1 -4303.071,E2 -4303.071} C_VEL
LIN {X 0,Y 531.006,Z 313.338,A -85,B 0,C 180,E1 -4305.435,E2 -4305.435} C_VEL
LIN {X 0,Y 531.029,Z 313.338,A -85,B 0,C 180,E1 -4308.549,E2 -4308.549} C_VEL
LIN {X 0,Y 531.051,Z 313.337,A -85,B 0,C 180,E1 -4311.629,E2 -4311.629} C_VEL
LIN {X 0,Y 531.12,Z 313.329,A -85,B 0,C 180,E1 -4314.685,E2 -4314.685} C_VEL
LIN {X 0,Y 531.135,Z 313.322,A -85,B 0,C 180,E1 -4317.725,E2 -4317.725} C_VEL
LIN {X 0,Y 531.136,Z 313.323,A -85,B 0,C 180,E1 -4320.758,E2 -4320.758} C_VEL
LIN {X 0,Y 531.094,Z 313.33,A -85,B 0,C 180,E1 -4323.034,E2 -4323.034} C_VEL
LIN {X 0,Y 531.088,Z 313.329,A -85,B 0,C 180,E1 -4326.077,E2 -4326.077} C_VEL
LIN {X 0,Y 531.03,Z 313.337,A -85,B 0,C 180,E1 -4329.138,E2 -4329.138} C_VEL
LIN {X 0,Y 531.018,Z 313.341,A -85,B 0,C 180,E1 -4332.225,E2 -4332.225} C_VEL
LIN {X 0,Y 530.985,Z 313.345,A -85,B 0,C 180,E1 -4335.35,E2 -4335.35} C_VEL
LIN {X 0,Y 530.984,Z 313.344,A -85,B 0,C 180,E1 -4338.521,E2 -4338.521} C_VEL
LIN {X 0,Y 530.998,Z 313.343,A -85,B 0,C 180,E1 -4340.938,E2 -4340.938} C_VEL
LIN {X 0,Y 530.969,Z 313.346,A -85,B 0,C 180,E1 -4344.225,E2 -4344.225} C_VEL
LIN {X 0,Y 530.963,Z 313.343,A -85,B 0,C 180,E1 -4346.746,E2 -4346.746} C_VEL
LIN {X 0,Y 530.956,Z 313.35,A -85,B 0,C 180,E1 -4349.324,E2 -4349.324} C_VEL
LIN {X 0,Y 530.967,Z 313.345,A -85,B 0,C 180,E1 -4352.102,E2 -4352.102} C_VEL
LIN {X 0,Y 530.981,Z 313.343,A -85,B 0,C 180,E1 -4354.854,E2 -4354.854} C_VEL
LIN {X 0,Y 530.963,Z 313.348,A -85,B 0,C 180,E1 -4357.508,E2 -4357.508} C_VEL
LIN {X 0,Y 530.95,Z 313.344,A -85,B 0,C 180,E1 -4360.436,E2 -4360.436} C_VEL
LIN {X 0,Y 530.932,Z 313.348,A -85,B 0,C 180,E1 -4363.498,E2 -4363.498} C_VEL
LIN {X 0,Y 530.953,Z 313.35,A -85,B 0,C 180,E1 -4366.505,E2 -4366.505} C_VEL
LIN {X 0,Y 530.985,Z 313.342,A -85,B 0,C 180,E1 -4368.977,E2 -4368.977} C_VEL
LIN {X 0,Y 530.954,Z 313.351,A -85,B 0,C 180,E1 -4371.53,E2 -4371.53} C_VEL
LIN {X 0,Y 531.019,Z 313.477,A -85,B 0,C 180,E1 -4372.638,E2 -4372.638} C_VEL
LIN {X 0,Y 531.557,Z 317.655,A -85,B 0,C 180,E1 -4374.427,E2 -4374.427} C_VEL
LIN {X 0,Y 531.486,Z 324.394,A -85,B 0,C 180,E1 -4377.17,E2 -4377.17} C_VEL
LIN {X 0,Y 531.338,Z 332.318,A -85,B 0,C 180,E1 -4380.264,E2 -4380.264} C_VEL
LIN {X 0,Y 531.143,Z 340.109,A -85,B 0,C 180,E1 -4383.264,E2 -4383.264} C_VEL
LIN {X 0,Y 531.037,Z 347.244,A -85,B 0,C 180,E1 -4385.949,E2 -4385.949} C_VEL
LIN {X 0,Y 530.926,Z 354.579,A -85,B 0,C 180,E1 -4388.653,E2 -4388.653} C_VEL
LIN {X 0,Y 530.802,Z 361.257,A -85,B 0,C 180,E1 -4391.072,E2 -4391.072} C_VEL
LIN {X 0,Y 530.71,Z 370.161,A -85,B 0,C 180,E1 -4394.248,E2 -4394.248} C_VEL
LIN {X 0,Y 530.623,Z 376.491,A -85,B 0,C 180,E1 -4396.476,E2 -4396.476} C_VEL
LIN {X 0,Y 532.327,Z 387.265,A -85,B 0,C 180,E1 -4396.763,E2 -4396.763} C_VEL
LIN {X 0,Y 532.125,Z 399.767,A -85,B 0,C 180,E1 -4397.17,E2 -4397.17} C_VEL
LIN {X 0,Y 531.857,Z 411.409,A -85,B 0,C 180,E1 -4397.697,E2 -4397.697} C_VEL
LIN {X 0,Y 531.652,Z 422.304,A -85,B 0,C 180,E1 -4398.34,E2 -4398.34} C_VEL
LIN {X 0,Y 531.395,Z 433.097,A -85,B 0,C 180,E1 -4399.137,E2 -4399.137} C_VEL
LIN {X 0,Y 531.114,Z 443.537,A -85,B 0,C 180,E1 -4400.094,E2 -4400.094} C_VEL
LIN {X 0,Y 530.931,Z 451.989,A -85,B 0,C 180,E1 -4401.052,E2 -4401.052} C_VEL
LIN {X 0,Y 530.758,Z 460.236,A -85,B 0,C 180,E1 -4402.199,E2 -4402.199} C_VEL
LIN {X 0,Y 530.598,Z 467.269,A -85,B 0,C 180,E1 -4403.419,E2 -4403.419} C_VEL
LIN {X 0,Y 530.524,Z 472.949,A -85,B 0,C 180,E1 -4404.679,E2 -4404.679} C_VEL
LIN {X 0,Y 530.523,Z 476.894,A -85,B 0,C 180,E1 -4405.821,E2 -4405.821} C_VEL
LIN {X 0,Y 530.457,Z 479.807,A -85,B 0,C 180,E1 -4406.962,E2 -4406.962} C_VEL
LIN {X 0,Y 530.411,Z 481.197,A -85,B 0,C 180,E1 -4407.722,E2 -4407.722} C_VEL
LIN {X 0,Y 530.344,Z 482.785,A -85,B 0,C 180,E1 -4409.24,E2 -4409.24} C_VEL
LIN {X 0,Y 530.342,Z 483,A -85,B 0,C 180,E1 -4410,E2 -4410} C_VEL
LIN {X 0,Y 530.361,Z 482.186,A -85,B 0,C 180,E1 -4411.518,E2 -4411.518} C_VEL
LIN {X 0,Y 530.411,Z 481.2,A -85,B 0,C 180,E1 -4412.278,E2 -4412.278} C_VEL
LIN {X 0,Y 530.457,Z 479.811,A -85,B 0,C 180,E1 -4413.037,E2 -4413.037} C_VEL
LIN {X 0,Y 530.522,Z 476.897,A -85,B 0,C 180,E1 -4414.178,E2 -4414.178} C_VEL
LIN {X 0,Y 530.524,Z 472.95,A -85,B 0,C 180,E1 -4415.32,E2 -4415.32} C_VEL
LIN {X 0,Y 530.598,Z 467.269,A -85,B 0,C 180,E1 -4416.581,E2 -4416.581} C_VEL
LIN {X 0,Y 530.758,Z 460.24,A -85,B 0,C 180,E1 -4417.8,E2 -4417.8} C_VEL
LIN {X 0,Y 530.93,Z 451.995,A -85,B 0,C 180,E1 -4418.947,E2 -4418.947} C_VEL
LIN {X 0,Y 531.112,Z 443.544,A -85,B 0,C 180,E1 -4419.905,E2 -4419.905} C_VEL
LIN {X 0,Y 531.406,Z 433.104,A -85,B 0,C 180,E1 -4420.862,E2 -4420.862} C_VEL
LIN {X 0,Y 531.64,Z 421.322,A -85,B 0,C 180,E1 -4421.727,E2 -4421.727} C_VEL
LIN {X 0,Y 531.913,Z 409.498,A -85,B 0,C 180,E1 -4422.398,E2 -4422.398} C_VEL
LIN {X 0,Y 532.153,Z 397.186,A -85,B 0,C 180,E1 -4422.925,E2 -4422.925} C_VEL
LIN {X 0,Y 532.204,Z 385.913,A -85,B 0,C 180,E1 -4423.276,E2 -4423.276} C_VEL
LIN {X 0,Y 530.622,Z 376.493,A -85,B 0,C 180,E1 -4423.523,E2 -4423.523} C_VEL
LIN {X 0,Y 530.715,Z 369.05,A -85,B 0,C 180,E1 -4426.146,E2 -4426.146} C_VEL
LIN {X 0,Y 530.848,Z 360.146,A -85,B 0,C 180,E1 -4429.328,E2 -4429.328} C_VEL
LIN {X 0,Y 530.976,Z 352.519,A -85,B 0,C 180,E1 -4432.101,E2 -4432.101} C_VEL
LIN {X 0,Y 531.089,Z 344.563,A -85,B 0,C 180,E1 -4435.052,E2 -4435.052} C_VEL
LIN {X 0,Y 531.211,Z 336.772,A -85,B 0,C 180,E1 -4438.012,E2 -4438.012} C_VEL
LIN {X 0,Y 531.376,Z 329.78,A -85,B 0,C 180,E1 -4440.718,E2 -4440.718} C_VEL
LIN {X 0,Y 531.537,Z 322.15,A -85,B 0,C 180,E1 -4443.732,E2 -4443.732} C_VEL
LIN {X 0,Y 531.582,Z 317.644,A -85,B 0,C 180,E1 -4445.57,E2 -4445.57} C_VEL
LIN {X 0,Y 531.004,Z 313.344,A -85,B 0,C 180,E1 -4447.503,E2 -4447.503} C_VEL
LIN {X 0,Y 531.022,Z 313.344,A -85,B 0,C 180,E1 -4450.428,E2 -4450.428} C_VEL
LIN {X 0,Y 530.961,Z 313.35,A -85,B 0,C 180,E1 -4453.493,E2 -4453.493} C_VEL
LIN {X 0,Y 530.978,Z 313.346,A -85,B 0,C 180,E1 -4455.62,E2 -4455.62} C_VEL
LIN {X 0,Y 530.955,Z 313.347,A -85,B 0,C 180,E1 -4458.561,E2 -4458.561} C_VEL
LIN {X 0,Y 530.949,Z 313.345,A -85,B 0,C 180,E1 -4461.528,E2 -4461.528} C_VEL
LIN {X 0,Y 530.975,Z 313.345,A -85,B 0,C 180,E1 -4464.381,E2 -4464.381} C_VEL
LIN {X 0,Y 530.963,Z 313.348,A -85,B 0,C 180,E1 -4467.133,E2 -4467.133} C_VEL
LIN {X 0,Y 530.942,Z 313.347,A -85,B 0,C 180,E1 -4469.801,E2 -4469.801} C_VEL
LIN {X 0,Y 530.958,Z 313.35,A -85,B 0,C 180,E1 -4472.476,E2 -4472.476} C_VEL
LIN {X 0,Y 530.979,Z 313.342,A -85,B 0,C 180,E1 -4474.941,E2 -4474.941} C_VEL
LIN {X 0,Y 530.968,Z 313.348,A -85,B 0,C 180,E1 -4477.897,E2 -4477.897} C_VEL
LIN {X 0,Y 530.987,Z 313.343,A -85,B 0,C 180,E1 -4480.677,E2 -4480.677} C_VEL
LIN {X 0,Y 530.968,Z 313.347,A -85,B 0,C 180,E1 -4483.07,E2 -4483.07} C_VEL
LIN {X 0,Y 530.995,Z 313.34,A -85,B 0,C 180,E1 -4485.435,E2 -4485.435} C_VEL
LIN {X 0,Y 531.024,Z 313.336,A -85,B 0,C 180,E1 -4488.549,E2 -4488.549} C_VEL
LIN {X 0,Y 531.05,Z 313.338,A -85,B 0,C 180,E1 -4491.629,E2 -4491.629} C_VEL
LIN {X 0,Y 531.133,Z 313.327,A -85,B 0,C 180,E1 -4494.685,E2 -4494.685} C_VEL
LIN {X 0,Y 531.13,Z 313.324,A -85,B 0,C 180,E1 -4497.725,E2 -4497.725} C_VEL
LIN {X 0,Y 531.132,Z 313.322,A -85,B 0,C 180,E1 -4500.758,E2 -4500.758} C_VEL
LIN {X 0,Y 531.092,Z 313.329,A -85,B 0,C 180,E1 -4503.034,E2 -4503.034} C_VEL
LIN {X 0,Y 531.084,Z 313.329,A -85,B 0,C 180,E1 -4506.077,E2 -4506.077} C_VEL
LIN {X 0,Y 531.025,Z 313.338,A -85,B 0,C 180,E1 -4509.138,E2 -4509.138} C_VEL
LIN {X 0,Y 531.014,Z 313.341,A -85,B 0,C 180,E1 -4512.226,E2 -4512.226} C_VEL
LIN {X 0,Y 530.981,Z 313.347,A -85,B 0,C 180,E1 -4515.35,E2 -4515.35} C_VEL
LIN {X 0,Y 530.983,Z 313.343,A -85,B 0,C 180,E1 -4518.522,E2 -4518.522} C_VEL
LIN {X 0,Y 530.993,Z 313.343,A -85,B 0,C 180,E1 -4520.938,E2 -4520.938} C_VEL
LIN {X 0,Y 530.963,Z 313.348,A -85,B 0,C 180,E1 -4524.225,E2 -4524.225} C_VEL
LIN {X 0,Y 530.974,Z 313.343,A -85,B 0,C 180,E1 -4526.745,E2 -4526.745} C_VEL
LIN {X 0,Y 530.951,Z 313.348,A -85,B 0,C 180,E1 -4529.325,E2 -4529.325} C_VEL
LIN {X 0,Y 530.963,Z 313.345,A -85,B 0,C 180,E1 -4532.102,E2 -4532.102} C_VEL
LIN {X 0,Y 530.982,Z 313.343,A -85,B 0,C 180,E1 -4534.855,E2 -4534.855} C_VEL
LIN {X 0,Y 530.959,Z 313.349,A -85,B 0,C 180,E1 -4537.508,E2 -4537.508} C_VEL
LIN {X 0,Y 530.947,Z 313.347,A -85,B 0,C 180,E1 -4540.436,E2 -4540.436} C_VEL
LIN {X 0,Y 530.93,Z 313.347,A -85,B 0,C 180,E1 -4543.572,E2 -4543.572} C_VEL
LIN {X 0,Y 530.266,Z 313.434,A -85,B 0,C 180,E1 -4544.206,E2 -4544.206} C_VEL
LIN {X 0,Y 527.426,Z 313.786,A -85,B 0,C 180,E1 -4545.235,E2 -4545.235} C_VEL
LIN {X 0,Y 525.027,Z 314.086,A -85,B 0,C 180,E1 -4546.064,E2 -4546.064} C_VEL
LIN {X 0,Y 523.997,Z 314.214,A -85,B 0,C 180,E1 -4546.704,E2 -4546.704} C_VEL
LIN {X 0,Y 523.913,Z 314.222,A -85,B 0,C 180,E1 -4546.92,E2 -4546.92} C_VEL
LIN {X 0,Y 523.975,Z 314.219,A -85,B 0,C 180,E1 -4549.924,E2 -4549.924} C_VEL
LIN {X 0,Y 523.899,Z 314.228,A -85,B 0,C 180,E1 -4552.868,E2 -4552.868} C_VEL
LIN {X 0,Y 523.825,Z 314.359,A -85,B 0,C 180,E1 -4554.767,E2 -4554.767} C_VEL
LIN {X 0,Y 523.836,Z 318.524,A -85,B 0,C 180,E1 -4557.545,E2 -4557.545} C_VEL
LIN {X 0,Y 523.73,Z 322.644,A -85,B 0,C 180,E1 -4560.232,E2 -4560.232} C_VEL
LIN {X 0,Y 523.647,Z 326.728,A -85,B 0,C 180,E1 -4562.851,E2 -4562.851} C_VEL
LIN {X 0,Y 523.646,Z 331.534,A -85,B 0,C 180,E1 -4565.874,E2 -4565.874} C_VEL
LIN {X 0,Y 523.504,Z 336.234,A -85,B 0,C 180,E1 -4568.749,E2 -4568.749} C_VEL
LIN {X 0,Y 523.471,Z 340.319,A -85,B 0,C 180,E1 -4571.204,E2 -4571.204} C_VEL
LIN {X 0,Y 523.408,Z 344.368,A -85,B 0,C 180,E1 -4573.623,E2 -4573.623} C_VEL
LIN {X 0,Y 523.425,Z 348.791,A -85,B 0,C 180,E1 -4576.213,E2 -4576.213} C_VEL
LIN {X 0,Y 523.428,Z 349.2,A -85,B 0,C 180,E1 -4576.374,E2 -4576.374} C_VEL
LIN {X 0,Y 525.359,Z 360.601,A -85,B 0,C 180,E1 -4576.708,E2 -4576.708} C_VEL
LIN {X 0,Y 525.114,Z 373.846,A -85,B 0,C 180,E1 -4577.194,E2 -4577.194} C_VEL
LIN {X 0,Y 524.851,Z 386.36,A -85,B 0,C 180,E1 -4577.825,E2 -4577.825} C_VEL
LIN {X 0,Y 524.597,Z 398.049,A -85,B 0,C 180,E1 -4578.604,E2 -4578.604} C_VEL
LIN {X 0,Y 524.308,Z 408.522,A -85,B 0,C 180,E1 -4579.477,E2 -4579.477} C_VEL
LIN {X 0,Y 524.062,Z 417.078,A -85,B 0,C 180,E1 -4580.35,E2 -4580.35} C_VEL
LIN {X 0,Y 523.868,Z 424.956,A -85,B 0,C 180,E1 -4581.32,E2 -4581.32} C_VEL
LIN {X 0,Y 523.659,Z 432.662,A -85,B 0,C 180,E1 -4582.482,E2 -4582.482} C_VEL
LIN {X 0,Y 523.543,Z 439.725,A -85,B 0,C 180,E1 -4583.835,E2 -4583.835} C_VEL
LIN {X 0,Y 523.383,Z 444.436,A -85,B 0,C 180,E1 -4584.993,E2 -4584.993} C_VEL
LIN {X 0,Y 523.443,Z 448.039,A -85,B 0,C 180,E1 -4586.151,E2 -4586.151} C_VEL
LIN {X 0,Y 523.367,Z 449.905,A -85,B 0,C 180,E1 -4586.921,E2 -4586.921} C_VEL
LIN {X 0,Y 523.335,Z 451.313,A -85,B 0,C 180,E1 -4587.691,E2 -4587.691} C_VEL
LIN {X 0,Y 523.25,Z 452.931,A -85,B 0,C 180,E1 -4589.231,E2 -4589.231} C_VEL
LIN {X 0,Y 523.247,Z 453.169,A -85,B 0,C 180,E1 -4590,E2 -4590} C_VEL
LIN {X 0,Y 523.25,Z 452.986,A -85,B 0,C 180,E1 -4590.77,E2 -4590.77} C_VEL
LIN {X 0,Y 523.336,Z 451.439,A -85,B 0,C 180,E1 -4592.309,E2 -4592.309} C_VEL
LIN {X 0,Y 523.368,Z 450.086,A -85,B 0,C 180,E1 -4593.079,E2 -4593.079} C_VEL
LIN {X 0,Y 523.442,Z 447.226,A -85,B 0,C 180,E1 -4594.235,E2 -4594.235} C_VEL
LIN {X 0,Y 523.463,Z 443.348,A -85,B 0,C 180,E1 -4595.393,E2 -4595.393} C_VEL
LIN {X 0,Y 523.526,Z 438.2,A -85,B 0,C 180,E1 -4596.583,E2 -4596.583} C_VEL
LIN {X 0,Y 523.671,Z 432.046,A -85,B 0,C 180,E1 -4597.713,E2 -4597.713} C_VEL
LIN {X 0,Y 523.884,Z 424.158,A -85,B 0,C 180,E1 -4598.875,E2 -4598.875} C_VEL
LIN {X 0,Y 524.118,Z 414.344,A -85,B 0,C 180,E1 -4600.039,E2 -4600.039} C_VEL
LIN {X 0,Y 524.411,Z 404.052,A -85,B 0,C 180,E1 -4601.01,E2 -4601.01} C_VEL
LIN {X 0,Y 524.675,Z 393.323,A -85,B 0,C 180,E1 -4601.824,E2 -4601.824} C_VEL
LIN {X 0,Y 524.899,Z 382.701,A -85,B 0,C 180,E1 -4602.469,E2 -4602.469} C_VEL
LIN {X 0,Y 525.247,Z 370.174,A -85,B 0,C 180,E1 -4603.05,E2 -4603.05} C_VEL
LIN {X 0,Y 525.236,Z 359.128,A -85,B 0,C 180,E1 -4603.428,E2 -4603.428} C_VEL
LIN {X 0,Y 523.418,Z 349.032,A -85,B 0,C 180,E1 -4603.739,E2 -4603.739} C_VEL
LIN {X 0,Y 523.401,Z 344.581,A -85,B 0,C 180,E1 -4606.378,E2 -4606.378} C_VEL
LIN {X 0,Y 523.462,Z 340.472,A -85,B 0,C 180,E1 -4608.797,E2 -4608.797} C_VEL
LIN {X 0,Y 523.506,Z 336.381,A -85,B 0,C 180,E1 -4611.252,E2 -4611.252} C_VEL
LIN {X 0,Y 523.636,Z 331.686,A -85,B 0,C 180,E1 -4614.123,E2 -4614.123} C_VEL
LIN {X 0,Y 523.648,Z 326.87,A -85,B 0,C 180,E1 -4617.15,E2 -4617.15} C_VEL
LIN {X 0,Y 523.719,Z 322.786,A -85,B 0,C 180,E1 -4619.77,E2 -4619.77} C_VEL
LIN {X 0,Y 523.835,Z 318.675,A -85,B 0,C 180,E1 -4622.456,E2 -4622.456} C_VEL
LIN {X 0,Y 523.866,Z 314.498,A -85,B 0,C 180,E1 -4625.23,E2 -4625.23} C_VEL
LIN {X 0,Y 523.905,Z 314.224,A -85,B 0,C 180,E1 -4627.677,E2 -4627.677} C_VEL
LIN {X 0,Y 523.937,Z 314.223,A -85,B 0,C 180,E1 -4630.129,E2 -4630.129} C_VEL
LIN {X 0,Y 523.937,Z 314.221,A -85,B 0,C 180,E1 -4632.459,E2 -4632.459} C_VEL
LIN {X 0,Y 523.94,Z 314.222,A -85,B 0,C 180,E1 -4635.31,E2 -4635.31} C_VEL
LIN {X 0,Y 523.917,Z 314.224,A -85,B 0,C 180,E1 -4638.694,E2 -4638.694} C_VEL
LIN {X 0,Y 523.911,Z 314.225,A -85,B 0,C 180,E1 -4641.898,E2 -4641.898} C_VEL
LIN {X 0,Y 523.933,Z 314.22,A -85,B 0,C 180,E1 -4644.909,E2 -4644.909} C_VEL
LIN {X 0,Y 523.935,Z 314.222,A -85,B 0,C 180,E1 -4647.679,E2 -4647.679} C_VEL
LIN {X 0,Y 523.931,Z 314.222,A -85,B 0,C 180,E1 -4650.68,E2 -4650.68} C_VEL
LIN {X 0,Y 523.904,Z 314.224,A -85,B 0,C 180,E1 -4653.725,E2 -4653.725} C_VEL
LIN {X 0,Y 523.905,Z 314.228,A -85,B 0,C 180,E1 -4656.269,E2 -4656.269} C_VEL
LIN {X 0,Y 523.943,Z 314.219,A -85,B 0,C 180,E1 -4658.766,E2 -4658.766} C_VEL
LIN {X 0,Y 523.946,Z 314.223,A -85,B 0,C 180,E1 -4661.22,E2 -4661.22} C_VEL
LIN {X 0,Y 523.926,Z 314.219,A -85,B 0,C 180,E1 -4663.638,E2 -4663.638} C_VEL
LIN {X 0,Y 523.916,Z 314.224,A -85,B 0,C 180,E1 -4666.027,E2 -4666.027} C_VEL
LIN {X 0,Y 523.989,Z 314.214,A -85,B 0,C 180,E1 -4669.177,E2 -4669.177} C_VEL
LIN {X 0,Y 524.024,Z 314.209,A -85,B 0,C 180,E1 -4672.292,E2 -4672.292} C_VEL
LIN {X 0,Y 524.082,Z 314.204,A -85,B 0,C 180,E1 -4674.614,E2 -4674.614} C_VEL
LIN {X 0,Y 524.106,Z 314.197,A -85,B 0,C 180,E1 -4677.694,E2 -4677.694} C_VEL
LIN {X 0,Y 524.086,Z 314.201,A -85,B 0,C 180,E1 -4680.768,E2 -4680.768} C_VEL
LIN {X 0,Y 524.062,Z 314.206,A -85,B 0,C 180,E1 -4683.075,E2 -4683.075} C_VEL
LIN {X 0,Y 524.049,Z 314.206,A -85,B 0,C 180,E1 -4686.159,E2 -4686.159} C_VEL
LIN {X 0,Y 523.997,Z 314.212,A -85,B 0,C 180,E1 -4689.262,E2 -4689.262} C_VEL
LIN {X 0,Y 523.993,Z 314.214,A -85,B 0,C 180,E1 -4691.737,E2 -4691.737} C_VEL
LIN {X 0,Y 523.977,Z 314.216,A -85,B 0,C 180,E1 -4695.048,E2 -4695.048} C_VEL
LIN {X 0,Y 523.959,Z 314.217,A -85,B 0,C 180,E1 -4697.969,E2 -4697.969} C_VEL
LIN {X 0,Y 523.968,Z 314.22,A -85,B 0,C 180,E1 -4700.41,E2 -4700.41} C_VEL
LIN {X 0,Y 523.913,Z 314.223,A -85,B 0,C 180,E1 -4702.894,E2 -4702.894} C_VEL
LIN {X 0,Y 523.922,Z 314.223,A -85,B 0,C 180,E1 -4705.42,E2 -4705.42} C_VEL
LIN {X 0,Y 523.9,Z 314.224,A -85,B 0,C 180,E1 -4708.003,E2 -4708.003} C_VEL
LIN {X 0,Y 523.932,Z 314.224,A -85,B 0,C 180,E1 -4710.853,E2 -4710.853} C_VEL
LIN {X 0,Y 523.958,Z 314.218,A -85,B 0,C 180,E1 -4713.735,E2 -4713.735} C_VEL
LIN {X 0,Y 523.919,Z 314.224,A -85,B 0,C 180,E1 -4716.404,E2 -4716.404} C_VEL
LIN {X 0,Y 523.915,Z 314.224,A -85,B 0,C 180,E1 -4719.085,E2 -4719.085} C_VEL
LIN {X 0,Y 523.896,Z 314.224,A -85,B 0,C 180,E1 -4722.125,E2 -4722.125} C_VEL
LIN {X 0,Y 523.939,Z 314.22,A -85,B 0,C 180,E1 -4725.311,E2 -4725.311} C_VEL
LIN {X 0,Y 523.958,Z 314.218,A -85,B 0,C 180,E1 -4728.69,E2 -4728.69} C_VEL
LIN {X 0,Y 523.921,Z 314.227,A -85,B 0,C 180,E1 -4731.899,E2 -4731.899} C_VEL
LIN {X 0,Y 523.982,Z 314.344,A -85,B 0,C 180,E1 -4732.462,E2 -4732.462} C_VEL
LIN {X 0,Y 524.559,Z 318.682,A -85,B 0,C 180,E1 -4734.353,E2 -4734.353} C_VEL
LIN {X 0,Y 524.498,Z 325.441,A -85,B 0,C 180,E1 -4737.134,E2 -4737.134} C_VEL
LIN {X 0,Y 524.309,Z 333.384,A -85,B 0,C 180,E1 -4740.267,E2 -4740.267} C_VEL
LIN {X 0,Y 524.172,Z 340.109,A -85,B 0,C 180,E1 -4742.88,E2 -4742.88} C_VEL
LIN {X 0,Y 524.009,Z 347.72,A -85,B 0,C 180,E1 -4745.786,E2 -4745.786} C_VEL
LIN {X 0,Y 523.864,Z 355.692,A -85,B 0,C 180,E1 -4748.763,E2 -4748.763} C_VEL
LIN {X 0,Y 523.725,Z 363.483,A -85,B 0,C 180,E1 -4751.618,E2 -4751.618} C_VEL
LIN {X 0,Y 523.658,Z 371.274,A -85,B 0,C 180,E1 -4754.43,E2 -4754.43} C_VEL
LIN {X 0,Y 523.557,Z 376.491,A -85,B 0,C 180,E1 -4756.29,E2 -4756.29} C_VEL
LIN {X 0,Y 525.387,Z 388.179,A -85,B 0,C 180,E1 -4756.609,E2 -4756.609} C_VEL
LIN {X 0,Y 525.184,Z 400.982,A -85,B 0,C 180,E1 -4757.047,E2 -4757.047} C_VEL
LIN {X 0,Y 524.89,Z 413.174,A -85,B 0,C 180,E1 -4757.629,E2 -4757.629} C_VEL
LIN {X 0,Y 524.649,Z 424.132,A -85,B 0,C 180,E1 -4758.307,E2 -4758.307} C_VEL
LIN {X 0,Y 524.362,Z 435.399,A -85,B 0,C 180,E1 -4759.185,E2 -4759.185} C_VEL
LIN {X 0,Y 524.086,Z 445.334,A -85,B 0,C 180,E1 -4760.155,E2 -4760.155} C_VEL
LIN {X 0,Y 523.852,Z 454.959,A -85,B 0,C 180,E1 -4761.319,E2 -4761.319} C_VEL
LIN {X 0,Y 523.633,Z 462.62,A -85,B 0,C 180,E1 -4762.48,E2 -4762.48} C_VEL
LIN {X 0,Y 523.515,Z 469.679,A -85,B 0,C 180,E1 -4763.834,E2 -4763.834} C_VEL
LIN {X 0,Y 523.384,Z 474.371,A -85,B 0,C 180,E1 -4764.992,E2 -4764.992} C_VEL
LIN {X 0,Y 523.443,Z 477.957,A -85,B 0,C 180,E1 -4766.15,E2 -4766.15} C_VEL
LIN {X 0,Y 523.367,Z 479.807,A -85,B 0,C 180,E1 -4766.921,E2 -4766.921} C_VEL
LIN {X 0,Y 523.335,Z 481.196,A -85,B 0,C 180,E1 -4767.691,E2 -4767.691} C_VEL
LIN {X 0,Y 523.25,Z 482.785,A -85,B 0,C 180,E1 -4769.23,E2 -4769.23} C_VEL
LIN {X 0,Y 523.246,Z 483,A -85,B 0,C 180,E1 -4770,E2 -4770} C_VEL
LIN {X 0,Y 523.275,Z 482.186,A -85,B 0,C 180,E1 -4771.539,E2 -4771.539} C_VEL
LIN {X 0,Y 523.335,Z 481.199,A -85,B 0,C 180,E1 -4772.309,E2 -4772.309} C_VEL
LIN {X 0,Y 523.367,Z 479.811,A -85,B 0,C 180,E1 -4773.079,E2 -4773.079} C_VEL
LIN {X 0,Y 523.441,Z 476.897,A -85,B 0,C 180,E1 -4774.234,E2 -4774.234} C_VEL
LIN {X 0,Y 523.464,Z 472.95,A -85,B 0,C 180,E1 -4775.392,E2 -4775.392} C_VEL
LIN {X 0,Y 523.522,Z 467.731,A -85,B 0,C 180,E1 -4776.58,E2 -4776.58} C_VEL
LIN {X 0,Y 523.664,Z 461.471,A -85,B 0,C 180,E1 -4777.712,E2 -4777.712} C_VEL
LIN {X 0,Y 523.856,Z 453.482,A -85,B 0,C 180,E1 -4778.875,E2 -4778.875} C_VEL
LIN {X 0,Y 524.085,Z 445.34,A -85,B 0,C 180,E1 -4779.844,E2 -4779.844} C_VEL
LIN {X 0,Y 524.364,Z 435.406,A -85,B 0,C 180,E1 -4780.815,E2 -4780.815} C_VEL
LIN {X 0,Y 524.628,Z 424.252,A -85,B 0,C 180,E1 -4781.685,E2 -4781.685} C_VEL
LIN {X 0,Y 524.849,Z 413.186,A -85,B 0,C 180,E1 -4782.371,E2 -4782.371} C_VEL
LIN {X 0,Y 525.167,Z 400.992,A -85,B 0,C 180,E1 -4782.953,E2 -4782.953} C_VEL
LIN {X 0,Y 525.417,Z 388.198,A -85,B 0,C 180,E1 -4783.389,E2 -4783.389} C_VEL
LIN {X 0,Y 523.556,Z 376.493,A -85,B 0,C 180,E1 -4783.71,E2 -4783.71} C_VEL
LIN {X 0,Y 523.643,Z 369.05,A -85,B 0,C 180,E1 -4786.37,E2 -4786.37} C_VEL
LIN {X 0,Y 523.805,Z 360.146,A -85,B 0,C 180,E1 -4789.598,E2 -4789.598} C_VEL
LIN {X 0,Y 523.916,Z 352.982,A -85,B 0,C 180,E1 -4792.242,E2 -4792.242} C_VEL
LIN {X 0,Y 524.056,Z 344.563,A -85,B 0,C 180,E1 -4795.412,E2 -4795.412} C_VEL
LIN {X 0,Y 524.205,Z 337.885,A -85,B 0,C 180,E1 -4797.984,E2 -4797.984} C_VEL
LIN {X 0,Y 524.338,Z 331.09,A -85,B 0,C 180,E1 -4800.618,E2 -4800.618} C_VEL
LIN {X 0,Y 524.549,Z 323.063,A -85,B 0,C 180,E1 -4803.83,E2 -4803.83} C_VEL
LIN {X 0,Y 524.578,Z 318.68,A -85,B 0,C 180,E1 -4805.645,E2 -4805.645} C_VEL
LIN {X 0,Y 523.938,Z 314.224,A -85,B 0,C 180,E1 -4807.682,E2 -4807.682} C_VEL
LIN {X 0,Y 523.964,Z 314.222,A -85,B 0,C 180,E1 -4810.133,E2 -4810.133} C_VEL
LIN {X 0,Y 523.92,Z 314.225,A -85,B 0,C 180,E1 -4813.165,E2 -4813.165} C_VEL
LIN {X 0,Y 523.93,Z 314.223,A -85,B 0,C 180,E1 -4815.771,E2 -4815.771} C_VEL
LIN {X 0,Y 523.892,Z 314.23,A -85,B 0,C 180,E1 -4818.903,E2 -4818.903} C_VEL
LIN {X 0,Y 523.908,Z 314.224,A -85,B 0,C 180,E1 -4821.897,E2 -4821.897} C_VEL
LIN {X 0,Y 523.931,Z 314.221,A -85,B 0,C 180,E1 -4824.908,E2 -4824.908} C_VEL
LIN {X 0,Y 523.93,Z 314.224,A -85,B 0,C 180,E1 -4827.678,E2 -4827.678} C_VEL
LIN {X 0,Y 523.925,Z 314.225,A -85,B 0,C 180,E1 -4830.68,E2 -4830.68} C_VEL
LIN {X 0,Y 523.926,Z 314.22,A -85,B 0,C 180,E1 -4833.726,E2 -4833.726} C_VEL
LIN {X 0,Y 523.926,Z 314.224,A -85,B 0,C 180,E1 -4836.27,E2 -4836.27} C_VEL
LIN {X 0,Y 523.938,Z 314.22,A -85,B 0,C 180,E1 -4838.766,E2 -4838.766} C_VEL
LIN {X 0,Y 523.944,Z 314.222,A -85,B 0,C 180,E1 -4841.22,E2 -4841.22} C_VEL
LIN {X 0,Y 523.918,Z 314.222,A -85,B 0,C 180,E1 -4843.638,E2 -4843.638} C_VEL
LIN {X 0,Y 523.913,Z 314.225,A -85,B 0,C 180,E1 -4846.027,E2 -4846.027} C_VEL
LIN {X 0,Y 523.985,Z 314.213,A -85,B 0,C 180,E1 -4849.177,E2 -4849.177} C_VEL
LIN {X 0,Y 524.019,Z 314.209,A -85,B 0,C 180,E1 -4852.292,E2 -4852.292} C_VEL
LIN {X 0,Y 524.092,Z 314.204,A -85,B 0,C 180,E1 -4854.614,E2 -4854.614} C_VEL
LIN {X 0,Y 524.102,Z 314.2,A -85,B 0,C 180,E1 -4857.694,E2 -4857.694} C_VEL
LIN {X 0,Y 524.103,Z 314.198,A -85,B 0,C 180,E1 -4860.768,E2 -4860.768} C_VEL
LIN {X 0,Y 524.06,Z 314.205,A -85,B 0,C 180,E1 -4863.075,E2 -4863.075} C_VEL
LIN {X 0,Y 524.044,Z 314.206,A -85,B 0,C 180,E1 -4866.159,E2 -4866.159} C_VEL
LIN {X 0,Y 523.992,Z 314.213,A -85,B 0,C 180,E1 -4869.262,E2 -4869.262} C_VEL
LIN {X 0,Y 523.988,Z 314.217,A -85,B 0,C 180,E1 -4871.738,E2 -4871.738} C_VEL
LIN {X 0,Y 523.975,Z 314.216,A -85,B 0,C 180,E1 -4875.05,E2 -4875.05} C_VEL
LIN {X 0,Y 523.954,Z 314.216,A -85,B 0,C 180,E1 -4877.969,E2 -4877.969} C_VEL
LIN {X 0,Y 523.963,Z 314.219,A -85,B 0,C 180,E1 -4880.411,E2 -4880.411} C_VEL
LIN {X 0,Y 523.908,Z 314.224,A -85,B 0,C 180,E1 -4882.894,E2 -4882.894} C_VEL
LIN {X 0,Y 523.92,Z 314.225,A -85,B 0,C 180,E1 -4885.421,E2 -4885.421} C_VEL
LIN {X 0,Y 523.898,Z 314.225,A -85,B 0,C 180,E1 -4888.003,E2 -4888.003} C_VEL
LIN {X 0,Y 523.928,Z 314.227,A -85,B 0,C 180,E1 -4890.854,E2 -4890.854} C_VEL
LIN {X 0,Y 523.954,Z 314.218,A -85,B 0,C 180,E1 -4893.736,E2 -4893.736} C_VEL
LIN {X 0,Y 523.916,Z 314.224,A -85,B 0,C 180,E1 -4896.405,E2 -4896.405} C_VEL
LIN {X 0,Y 523.913,Z 314.226,A -85,B 0,C 180,E1 -4899.086,E2 -4899.086} C_VEL
LIN {X 0,Y 523.901,Z 314.224,A -85,B 0,C 180,E1 -4902.124,E2 -4902.124} C_VEL
LIN {X 0,Y 523.938,Z 314.218,A -85,B 0,C 180,E1 -4905.311,E2 -4905.311} C_VEL
LIN {X 0,Y 523.913,Z 314.222,A -85,B 0,C 180,E1 -4906.92,E2 -4906.92} C_VEL
LIN {X 0,Y 523.253,Z 314.306,A -85,B 0,C 180,E1 -4907.562,E2 -4907.562} C_VEL
LIN {X 0,Y 520.426,Z 314.658,A -85,B 0,C 180,E1 -4908.604,E2 -4908.604} C_VEL
LIN {X 0,Y 518.028,Z 314.958,A -85,B 0,C 180,E1 -4909.443,E2 -4909.443} C_VEL
LIN {X 0,Y 516.988,Z 315.088,A -85,B 0,C 180,E1 -4910.091,E2 -4910.091} C_VEL
LIN {X 0,Y 516.898,Z 315.097,A -85,B 0,C 180,E1 -4910.31,E2 -4910.31} C_VEL
LIN {X 0,Y 516.842,Z 315.108,A -85,B 0,C 180,E1 -4913.349,E2 -4913.349} C_VEL
